KUKA KRL program: EPS_2_251806_MH04A_A_20260212042233.src

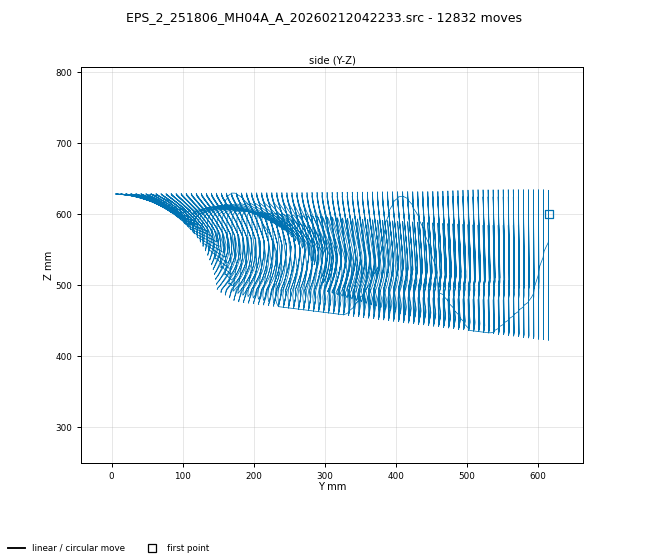
[picture p0: tool path of EPS_2_251806_MH04A_A_20260212042233.src, 12832 of 12834 moves have a stored position in this frame; points joined in program order, loops and branches not executed]
&ACCESS RVP
&REL 4
&COMMENT QRS 19112012
&PARAM EDITMASK = *
DEF PART()
EXT BAS (BAS_COMMAND :IN,REAL :IN )
INT I
BAS (#INITMOV,0 )

;KUKA QRS Post kuka4.cps  Date:22-06-2017 !

File_ID=3012

QRS_PRE_INIT()

;Init var - Until changes are made in qrs_pre_init
Outlet_Square_prg=0
Inlet_1_Square_prg=0
Inlet_2_Square_prg=0
Inlet_3_Square_prg=0
Inlet_4_Square_prg=0
Inlet_5_Square_prg=0

Outlet_1={X 0.000, Y 509.470, Z 509.000, B 0.000, E1 0.000 }
Inlet_1={X 0.000, Y 519.000, Z 484.000, B 0.000, E1 90.000 }
Inlet_2={X 0.000, Y 510.210, Z 499.000, B 0.000, E1 180.000 }
Outlet_1_type=251
Inlet_1_type=201
Inlet_2_type=251
;QRS#1=Sidecore dimensions
;QRS#2=250-10" PVC SDR 35
;QRS#3=200-8" PVC SDR 35
;QRS#4=250-10" PVC SDR 35
;QRS#5=
;QRS#6=
;QRS#7=
;QRS#8=
;QRS#9=14M PSX
;QRS#10=12-08 PSX
;QRS#11=14M PSX
;QRS#12=
;QRS#13=
;QRS#14=
;QRS#15=
;QRS#16=1220x127x914 3'
;QRS#17=EPS Height
;QRS#18=634,5
;QRS#19=*
;QRS#20= UPDATED VERSION 22-06-2017
;QRS#21=*
Outlet_Square=0100
Inlet_1_Square=0100
Inlet_2_Square=0100
Inlet_3_Square=0
Inlet_4_Square=0
Inlet_5_Square=0
Mill_Square=1
Outlet_Square_Prg=205
Inlet_1_Square_prg=204
Inlet_2_Square_prg=205

QRS_INIT()

$ADVANCE=5

; T1
PTP {E1 173.497,E2 173.497}
PTP {X 0,Y 615.499,A -85,B 0,C 180,E1 173.497,E2 173.497,E3 0,E4 0,E5 0,E6 0}
QRS_SPEED_INIT()
LIN {X 0,Y 615.499,Z 600,A -85,B 0,C 180,E1 173.497,E2 173.497,E3 0,E4 0,E5 0,E6 0} C_VEL
LIN {X 0,Y 615.499,Z 575.226,A -85,B 0,C 180,E1 173.497,E2 173.497} C_VEL
LIN {X 0,Y 615.499,Z 564.345,A -85,B 0,C 180,E1 173.497,E2 173.497} C_VEL
LIN {X 0,Y 615.497,Z 562.701,A -85,B 0,C 180,E1 173.417,E2 173.417} C_VEL
LIN {X 0,Y 615.497,Z 555.036,A -85,B 0,C 180,E1 172.455,E2 172.455} C_VEL
LIN {X 0,Y 615.498,Z 545.258,A -85,B 0,C 180,E1 171.463,E2 171.463} C_VEL
LIN {X 0,Y 615.498,Z 534.992,A -85,B 0,C 180,E1 170.636,E2 170.636} C_VEL
LIN {X 0,Y 615.481,Z 523.43,A -85,B 0,C 180,E1 169.889,E2 169.889} C_VEL
LIN {X 0,Y 615.482,Z 511.646,A -85,B 0,C 180,E1 169.296,E2 169.296} C_VEL
LIN {X 0,Y 615.483,Z 498.658,A -85,B 0,C 180,E1 168.807,E2 168.807} C_VEL
LIN {X 0,Y 615.487,Z 486.055,A -85,B 0,C 180,E1 168.473,E2 168.473} C_VEL
LIN {X 0,Y 615.484,Z 478.768,A -85,B 0,C 180,E1 168.327,E2 168.327} C_VEL
LIN {X 0,Y 615.493,Z 471.461,A -85,B 0,C 180,E1 165.451,E2 165.451} C_VEL
LIN {X 0,Y 615.491,Z 464.645,A -85,B 0,C 180,E1 162.729,E2 162.729} C_VEL
LIN {X 0,Y 615.479,Z 457.814,A -85,B 0,C 180,E1 159.967,E2 159.967} C_VEL
LIN {X 0,Y 615.493,Z 452.183,A -85,B 0,C 180,E1 157.654,E2 157.654} C_VEL
LIN {X 0,Y 615.476,Z 445.867,A -85,B 0,C 180,E1 155.008,E2 155.008} C_VEL
LIN {X 0,Y 615.481,Z 440.735,A -85,B 0,C 180,E1 152.822,E2 152.822} C_VEL
LIN {X 0,Y 615.484,Z 434.726,A -85,B 0,C 180,E1 150.207,E2 150.207} C_VEL
LIN {X 0,Y 615.486,Z 428.763,A -85,B 0,C 180,E1 147.542,E2 147.542} C_VEL
LIN {X 0,Y 615.49,Z 422.483,A -85,B 0,C 180,E1 144.685,E2 144.685} C_VEL
LIN {X 0,Y 615.485,Z 422.323,A -85,B 0,C 180,E1 141.931,E2 141.931} C_VEL
LIN {X 0,Y 615.492,Z 422.327,A -85,B 0,C 180,E1 139.394,E2 139.394} C_VEL
LIN {X 0,Y 615.497,Z 422.32,A -85,B 0,C 180,E1 136.756,E2 136.756} C_VEL
LIN {X 0,Y 615.485,Z 422.327,A -85,B 0,C 180,E1 133.997,E2 133.997} C_VEL
LIN {X 0,Y 615.481,Z 422.323,A -85,B 0,C 180,E1 131.093,E2 131.093} C_VEL
LIN {X 0,Y 615.486,Z 422.322,A -85,B 0,C 180,E1 128.905,E2 128.905} C_VEL
LIN {X 0,Y 615.496,Z 422.527,A -85,B 0,C 180,E1 127.626,E2 127.626} C_VEL
LIN {X 0,Y 615.498,Z 431.499,A -85,B 0,C 180,E1 124.702,E2 124.702} C_VEL
LIN {X 0,Y 615.477,Z 438.274,A -85,B 0,C 180,E1 122.329,E2 122.329} C_VEL
LIN {X 0,Y 615.498,Z 445.339,A -85,B 0,C 180,E1 119.796,E2 119.796} C_VEL
LIN {X 0,Y 615.486,Z 453.213,A -85,B 0,C 180,E1 117.044,E2 117.044} C_VEL
LIN {X 0,Y 615.478,Z 461.349,A -85,B 0,C 180,E1 114.273,E2 114.273} C_VEL
LIN {X 0,Y 615.48,Z 469.853,A -85,B 0,C 180,E1 111.433,E2 111.433} C_VEL
LIN {X 0,Y 615.481,Z 478.503,A -85,B 0,C 180,E1 108.602,E2 108.602} C_VEL
LIN {X 0,Y 615.488,Z 486.863,A -85,B 0,C 180,E1 105.906,E2 105.906} C_VEL
LIN {X 0,Y 615.494,Z 492.908,A -85,B 0,C 180,E1 103.993,E2 103.993} C_VEL
LIN {X 0,Y 615.492,Z 507.3,A -85,B 0,C 180,E1 103.748,E2 103.748} C_VEL
LIN {X 0,Y 615.479,Z 521.427,A -85,B 0,C 180,E1 103.37,E2 103.37} C_VEL
LIN {X 0,Y 615.495,Z 535.017,A -85,B 0,C 180,E1 102.866,E2 102.866} C_VEL
LIN {X 0,Y 615.479,Z 547.289,A -85,B 0,C 180,E1 102.28,E2 102.28} C_VEL
LIN {X 0,Y 615.498,Z 559.895,A -85,B 0,C 180,E1 101.527,E2 101.527} C_VEL
LIN {X 0,Y 615.498,Z 571.068,A -85,B 0,C 180,E1 100.709,E2 100.709} C_VEL
LIN {X 0,Y 615.499,Z 580.69,A -85,B 0,C 180,E1 99.863,E2 99.863} C_VEL
LIN {X 0,Y 615.497,Z 590.14,A -85,B 0,C 180,E1 98.868,E2 98.868} C_VEL
LIN {X 0,Y 615.497,Z 599.132,A -85,B 0,C 180,E1 97.711,E2 97.711} C_VEL
LIN {X 0,Y 615.496,Z 606.378,A -85,B 0,C 180,E1 96.557,E2 96.557} C_VEL
LIN {X 0,Y 615.491,Z 612.885,A -85,B 0,C 180,E1 95.242,E2 95.242} C_VEL
LIN {X 0,Y 615.496,Z 617.754,A -85,B 0,C 180,E1 93.929,E2 93.929} C_VEL
LIN {X 0,Y 615.496,Z 621.152,A -85,B 0,C 180,E1 92.619,E2 92.619} C_VEL
LIN {X 0,Y 615.493,Z 623.173,A -85,B 0,C 180,E1 91.309,E2 91.309} C_VEL
LIN {X 0,Y 615.494,Z 623.884,A -85,B 0,C 180,E1 90.001,E2 90.001} C_VEL
LIN {X 0,Y 615.49,Z 623.281,A -85,B 0,C 180,E1 88.692,E2 88.692} C_VEL
LIN {X 0,Y 615.493,Z 621.352,A -85,B 0,C 180,E1 87.383,E2 87.383} C_VEL
LIN {X 0,Y 615.496,Z 618.048,A -85,B 0,C 180,E1 86.072,E2 86.072} C_VEL
LIN {X 0,Y 615.496,Z 613.277,A -85,B 0,C 180,E1 84.76,E2 84.76} C_VEL
LIN {X 0,Y 615.494,Z 606.879,A -85,B 0,C 180,E1 83.444,E2 83.444} C_VEL
LIN {X 0,Y 615.496,Z 599.75,A -85,B 0,C 180,E1 82.29,E2 82.29} C_VEL
LIN {X 0,Y 615.497,Z 592.278,A -85,B 0,C 180,E1 81.299,E2 81.299} C_VEL
LIN {X 0,Y 615.495,Z 583.3,A -85,B 0,C 180,E1 80.305,E2 80.305} C_VEL
LIN {X 0,Y 615.499,Z 572.211,A -85,B 0,C 180,E1 79.291,E2 79.291} C_VEL
LIN {X 0,Y 615.498,Z 561.294,A -85,B 0,C 180,E1 78.474,E2 78.474} C_VEL
LIN {X 0,Y 615.483,Z 549.001,A -85,B 0,C 180,E1 77.722,E2 77.722} C_VEL
LIN {X 0,Y 615.495,Z 537.167,A -85,B 0,C 180,E1 77.136,E2 77.136} C_VEL
LIN {X 0,Y 615.475,Z 524.249,A -85,B 0,C 180,E1 76.631,E2 76.631} C_VEL
LIN {X 0,Y 615.484,Z 511.28,A -85,B 0,C 180,E1 76.253,E2 76.253} C_VEL
LIN {X 0,Y 615.494,Z 497.969,A -85,B 0,C 180,E1 75.987,E2 75.987} C_VEL
LIN {X 0,Y 615.489,Z 492.846,A -85,B 0,C 180,E1 75.911,E2 75.911} C_VEL
LIN {X 0,Y 615.491,Z 483.961,A -85,B 0,C 180,E1 73.073,E2 73.073} C_VEL
LIN {X 0,Y 615.488,Z 475.45,A -85,B 0,C 180,E1 70.316,E2 70.316} C_VEL
LIN {X 0,Y 615.477,Z 467.387,A -85,B 0,C 180,E1 67.657,E2 67.657} C_VEL
LIN {X 0,Y 615.488,Z 459.484,A -85,B 0,C 180,E1 65.009,E2 65.009} C_VEL
LIN {X 0,Y 615.488,Z 450.967,A -85,B 0,C 180,E1 62.086,E2 62.086} C_VEL
LIN {X 0,Y 615.477,Z 443.502,A -85,B 0,C 180,E1 59.462,E2 59.462} C_VEL
LIN {X 0,Y 615.492,Z 436.035,A -85,B 0,C 180,E1 56.765,E2 56.765} C_VEL
LIN {X 0,Y 615.493,Z 428.318,A -85,B 0,C 180,E1 54.166,E2 54.166} C_VEL
LIN {X 0,Y 615.498,Z 422.315,A -85,B 0,C 180,E1 52.183,E2 52.183} C_VEL
LIN {X 0,Y 615.484,Z 422.319,A -85,B 0,C 180,E1 49.395,E2 49.395} C_VEL
LIN {X 0,Y 615.476,Z 422.316,A -85,B 0,C 180,E1 46.756,E2 46.756} C_VEL
LIN {X 0,Y 615.488,Z 422.324,A -85,B 0,C 180,E1 43.999,E2 43.999} C_VEL
LIN {X 0,Y 615.485,Z 422.313,A -85,B 0,C 180,E1 41.474,E2 41.474} C_VEL
LIN {X 0,Y 615.481,Z 422.322,A -85,B 0,C 180,E1 38.905,E2 38.905} C_VEL
LIN {X 0,Y 615.493,Z 422.313,A -85,B 0,C 180,E1 36.425,E2 36.425} C_VEL
LIN {X 0,Y 615.496,Z 422.324,A -85,B 0,C 180,E1 33.538,E2 33.538} C_VEL
LIN {X 0,Y 615.478,Z 422.314,A -85,B 0,C 180,E1 30.92,E2 30.92} C_VEL
LIN {X 0,Y 615.491,Z 422.322,A -85,B 0,C 180,E1 28.454,E2 28.454} C_VEL
LIN {X 0,Y 615.484,Z 422.313,A -85,B 0,C 180,E1 25.571,E2 25.571} C_VEL
LIN {X 0,Y 615.489,Z 422.32,A -85,B 0,C 180,E1 22.845,E2 22.845} C_VEL
LIN {X 0,Y 615.487,Z 422.317,A -85,B 0,C 180,E1 20.033,E2 20.033} C_VEL
LIN {X 0,Y 615.489,Z 422.313,A -85,B 0,C 180,E1 17.271,E2 17.271} C_VEL
LIN {X 0,Y 615.49,Z 422.323,A -85,B 0,C 180,E1 14.549,E2 14.549} C_VEL
LIN {X 0,Y 615.478,Z 422.314,A -85,B 0,C 180,E1 11.861,E2 11.861} C_VEL
LIN {X 0,Y 615.497,Z 422.325,A -85,B 0,C 180,E1 9.199,E2 9.199} C_VEL
LIN {X 0,Y 615.492,Z 422.311,A -85,B 0,C 180,E1 6.557,E2 6.557} C_VEL
LIN {X 0,Y 615.488,Z 422.324,A -85,B 0,C 180,E1 3.929,E2 3.929} C_VEL
LIN {X 0,Y 615.486,Z 422.313,A -85,B 0,C 180,E1 1.309,E2 1.309} C_VEL
LIN {X 0,Y 615.494,Z 422.322,A -85,B 0,C 180,E1 -1.309,E2 -1.309} C_VEL
LIN {X 0,Y 615.476,Z 422.315,A -85,B 0,C 180,E1 -3.929,E2 -3.929} C_VEL
LIN {X 0,Y 615.49,Z 422.32,A -85,B 0,C 180,E1 -6.592,E2 -6.592} C_VEL
LIN {X 0,Y 615.479,Z 422.315,A -85,B 0,C 180,E1 -9.199,E2 -9.199} C_VEL
LIN {X 0,Y 615.478,Z 422.321,A -85,B 0,C 180,E1 -11.861,E2 -11.861} C_VEL
LIN {X 0,Y 615.49,Z 422.315,A -85,B 0,C 180,E1 -14.549,E2 -14.549} C_VEL
LIN {X 0,Y 615.494,Z 422.313,A -85,B 0,C 180,E1 -17.27,E2 -17.27} C_VEL
LIN {X 0,Y 615.489,Z 422.321,A -85,B 0,C 180,E1 -20.033,E2 -20.033} C_VEL
LIN {X 0,Y 615.476,Z 422.315,A -85,B 0,C 180,E1 -22.845,E2 -22.845} C_VEL
LIN {X 0,Y 615.486,Z 422.323,A -85,B 0,C 180,E1 -25.571,E2 -25.571} C_VEL
LIN {X 0,Y 615.492,Z 422.315,A -85,B 0,C 180,E1 -28.454,E2 -28.454} C_VEL
LIN {X 0,Y 615.49,Z 422.315,A -85,B 0,C 180,E1 -31.089,E2 -31.089} C_VEL
LIN {X 0,Y 615.489,Z 422.314,A -85,B 0,C 180,E1 -33.537,E2 -33.537} C_VEL
LIN {X 0,Y 615.488,Z 422.313,A -85,B 0,C 180,E1 -36.425,E2 -36.425} C_VEL
LIN {X 0,Y 615.481,Z 422.322,A -85,B 0,C 180,E1 -39.063,E2 -39.063} C_VEL
LIN {X 0,Y 615.485,Z 422.316,A -85,B 0,C 180,E1 -41.474,E2 -41.474} C_VEL
LIN {X 0,Y 615.491,Z 422.317,A -85,B 0,C 180,E1 -44.149,E2 -44.149} C_VEL
LIN {X 0,Y 615.481,Z 422.314,A -85,B 0,C 180,E1 -46.953,E2 -46.953} C_VEL
LIN {X 0,Y 615.492,Z 422.318,A -85,B 0,C 180,E1 -49.395,E2 -49.395} C_VEL
LIN {X 0,Y 615.484,Z 422.315,A -85,B 0,C 180,E1 -51.989,E2 -51.989} C_VEL
LIN {X 0,Y 615.487,Z 422.315,A -85,B 0,C 180,E1 -54.386,E2 -54.386} C_VEL
LIN {X 0,Y 615.494,Z 422.321,A -85,B 0,C 180,E1 -56.766,E2 -56.766} C_VEL
LIN {X 0,Y 615.484,Z 422.445,A -85,B 0,C 180,E1 -57.954,E2 -57.954} C_VEL
LIN {X 0,Y 615.477,Z 433.27,A -85,B 0,C 180,E1 -60.594,E2 -60.594} C_VEL
LIN {X 0,Y 615.495,Z 444.461,A -85,B 0,C 180,E1 -63.257,E2 -63.257} C_VEL
LIN {X 0,Y 615.482,Z 456.236,A -85,B 0,C 180,E1 -65.993,E2 -65.993} C_VEL
LIN {X 0,Y 615.477,Z 467.542,A -85,B 0,C 180,E1 -68.569,E2 -68.569} C_VEL
LIN {X 0,Y 615.481,Z 480.178,A -85,B 0,C 180,E1 -71.397,E2 -71.397} C_VEL
LIN {X 0,Y 615.485,Z 492.418,A -85,B 0,C 180,E1 -74.096,E2 -74.096} C_VEL
LIN {X 0,Y 615.489,Z 500.83,A -85,B 0,C 180,E1 -75.93,E2 -75.93} C_VEL
LIN {X 0,Y 615.492,Z 515.627,A -85,B 0,C 180,E1 -76.169,E2 -76.169} C_VEL
LIN {X 0,Y 615.486,Z 528.953,A -85,B 0,C 180,E1 -76.506,E2 -76.506} C_VEL
LIN {X 0,Y 615.492,Z 542.169,A -85,B 0,C 180,E1 -76.968,E2 -76.968} C_VEL
LIN {X 0,Y 615.478,Z 555.035,A -85,B 0,C 180,E1 -77.554,E2 -77.554} C_VEL
LIN {X 0,Y 615.497,Z 566.787,A -85,B 0,C 180,E1 -78.224,E2 -78.224} C_VEL
LIN {X 0,Y 615.496,Z 577.419,A -85,B 0,C 180,E1 -78.958,E2 -78.958} C_VEL
LIN {X 0,Y 615.498,Z 587.651,A -85,B 0,C 180,E1 -79.807,E2 -79.807} C_VEL
LIN {X 0,Y 615.498,Z 597.595,A -85,B 0,C 180,E1 -80.802,E2 -80.802} C_VEL
LIN {X 0,Y 615.496,Z 607.079,A -85,B 0,C 180,E1 -81.96,E2 -81.96} C_VEL
LIN {X 0,Y 615.495,Z 614.656,A -85,B 0,C 180,E1 -83.101,E2 -83.101} C_VEL
LIN {X 0,Y 615.494,Z 620.075,A -85,B 0,C 180,E1 -84.102,E2 -84.102} C_VEL
LIN {X 0,Y 615.495,Z 625.686,A -85,B 0,C 180,E1 -85.416,E2 -85.416} C_VEL
LIN {X 0,Y 615.495,Z 629.756,A -85,B 0,C 180,E1 -86.728,E2 -86.728} C_VEL
LIN {X 0,Y 615.497,Z 632.407,A -85,B 0,C 180,E1 -88.038,E2 -88.038} C_VEL
LIN {X 0,Y 615.493,Z 633.723,A -85,B 0,C 180,E1 -89.347,E2 -89.347} C_VEL
LIN {X 0,Y 615.493,Z 633.722,A -85,B 0,C 180,E1 -90.655,E2 -90.655} C_VEL
LIN {X 0,Y 615.498,Z 632.404,A -85,B 0,C 180,E1 -91.964,E2 -91.964} C_VEL
LIN {X 0,Y 615.495,Z 629.752,A -85,B 0,C 180,E1 -93.274,E2 -93.274} C_VEL
LIN {X 0,Y 615.495,Z 625.68,A -85,B 0,C 180,E1 -94.585,E2 -94.585} C_VEL
LIN {X 0,Y 615.494,Z 620.066,A -85,B 0,C 180,E1 -95.899,E2 -95.899} C_VEL
LIN {X 0,Y 615.495,Z 614.651,A -85,B 0,C 180,E1 -96.9,E2 -96.9} C_VEL
LIN {X 0,Y 615.496,Z 607.067,A -85,B 0,C 180,E1 -98.041,E2 -98.041} C_VEL
LIN {X 0,Y 615.498,Z 597.58,A -85,B 0,C 180,E1 -99.199,E2 -99.199} C_VEL
LIN {X 0,Y 615.498,Z 587.633,A -85,B 0,C 180,E1 -100.195,E2 -100.195} C_VEL
LIN {X 0,Y 615.498,Z 576.377,A -85,B 0,C 180,E1 -101.118,E2 -101.118} C_VEL
LIN {X 0,Y 615.496,Z 565.403,A -85,B 0,C 180,E1 -101.861,E2 -101.861} C_VEL
LIN {X 0,Y 615.479,Z 553.314,A -85,B 0,C 180,E1 -102.531,E2 -102.531} C_VEL
LIN {X 0,Y 615.488,Z 539.91,A -85,B 0,C 180,E1 -103.118,E2 -103.118} C_VEL
LIN {X 0,Y 615.488,Z 525.869,A -85,B 0,C 180,E1 -103.58,E2 -103.58} C_VEL
LIN {X 0,Y 615.496,Z 511.604,A -85,B 0,C 180,E1 -103.905,E2 -103.905} C_VEL
LIN {X 0,Y 615.489,Z 500.829,A -85,B 0,C 180,E1 -104.07,E2 -104.07} C_VEL
LIN {X 0,Y 615.494,Z 487.748,A -85,B 0,C 180,E1 -106.929,E2 -106.929} C_VEL
LIN {X 0,Y 615.487,Z 475.313,A -85,B 0,C 180,E1 -109.686,E2 -109.686} C_VEL
LIN {X 0,Y 615.487,Z 462.409,A -85,B 0,C 180,E1 -112.594,E2 -112.594} C_VEL
LIN {X 0,Y 615.477,Z 450.731,A -85,B 0,C 180,E1 -115.28,E2 -115.28} C_VEL
LIN {X 0,Y 615.493,Z 439.498,A -85,B 0,C 180,E1 -117.915,E2 -117.915} C_VEL
LIN {X 0,Y 615.479,Z 428.584,A -85,B 0,C 180,E1 -120.54,E2 -120.54} C_VEL
LIN {X 0,Y 615.482,Z 422.32,A -85,B 0,C 180,E1 -122.087,E2 -122.087} C_VEL
LIN {X 0,Y 615.499,Z 422.319,A -85,B 0,C 180,E1 -124.815,E2 -124.815} C_VEL
LIN {X 0,Y 615.488,Z 422.321,A -85,B 0,C 180,E1 -127.243,E2 -127.243} C_VEL
LIN {X 0,Y 615.483,Z 422.321,A -85,B 0,C 180,E1 -130.088,E2 -130.088} C_VEL
LIN {X 0,Y 615.491,Z 422.319,A -85,B 0,C 180,E1 -133.048,E2 -133.048} C_VEL
LIN {X 0,Y 615.488,Z 422.32,A -85,B 0,C 180,E1 -136.003,E2 -136.003} C_VEL
LIN {X 0,Y 615.492,Z 422.319,A -85,B 0,C 180,E1 -138.906,E2 -138.906} C_VEL
LIN {X 0,Y 615.49,Z 422.321,A -85,B 0,C 180,E1 -141.932,E2 -141.932} C_VEL
LIN {X 0,Y 615.495,Z 422.386,A -85,B 0,C 180,E1 -144.886,E2 -144.886} C_VEL
LIN {X 0,Y 615.493,Z 428.829,A -85,B 0,C 180,E1 -147.669,E2 -147.669} C_VEL
LIN {X 0,Y 615.492,Z 435.398,A -85,B 0,C 180,E1 -150.594,E2 -150.594} C_VEL
LIN {X 0,Y 615.48,Z 440.839,A -85,B 0,C 180,E1 -152.957,E2 -152.957} C_VEL
LIN {X 0,Y 615.493,Z 447.354,A -85,B 0,C 180,E1 -155.728,E2 -155.728} C_VEL
LIN {X 0,Y 615.494,Z 454.183,A -85,B 0,C 180,E1 -158.568,E2 -158.568} C_VEL
LIN {X 0,Y 615.484,Z 461.112,A -85,B 0,C 180,E1 -161.397,E2 -161.397} C_VEL
LIN {X 0,Y 615.476,Z 467.832,A -85,B 0,C 180,E1 -164.095,E2 -164.095} C_VEL
LIN {X 0,Y 615.497,Z 474.644,A -85,B 0,C 180,E1 -166.799,E2 -166.799} C_VEL
LIN {X 0,Y 615.485,Z 478.804,A -85,B 0,C 180,E1 -168.431,E2 -168.431} C_VEL
LIN {X 0,Y 615.495,Z 491.197,A -85,B 0,C 180,E1 -168.682,E2 -168.682} C_VEL
LIN {X 0,Y 615.48,Z 503.99,A -85,B 0,C 180,E1 -169.079,E2 -169.079} C_VEL
LIN {X 0,Y 615.498,Z 515.321,A -85,B 0,C 180,E1 -169.556,E2 -169.556} C_VEL
LIN {X 0,Y 615.479,Z 526.127,A -85,B 0,C 180,E1 -170.138,E2 -170.138} C_VEL
LIN {X 0,Y 615.498,Z 537.159,A -85,B 0,C 180,E1 -170.884,E2 -170.884} C_VEL
LIN {X 0,Y 615.498,Z 547.831,A -85,B 0,C 180,E1 -171.794,E2 -171.794} C_VEL
LIN {X 0,Y 615.498,Z 555.709,A -85,B 0,C 180,E1 -172.62,E2 -172.62} C_VEL
LIN {X 0,Y 615.497,Z 563.399,A -85,B 0,C 180,E1 -173.608,E2 -173.608} C_VEL
LIN {X 0,Y 615.498,Z 570.458,A -85,B 0,C 180,E1 -174.759,E2 -174.759} C_VEL
LIN {X 0,Y 615.493,Z 575.158,A -85,B 0,C 180,E1 -175.744,E2 -175.744} C_VEL
LIN {X 0,Y 615.496,Z 578.754,A -85,B 0,C 180,E1 -176.727,E2 -176.727} C_VEL
LIN {X 0,Y 615.496,Z 580.615,A -85,B 0,C 180,E1 -177.382,E2 -177.382} C_VEL
LIN {X 0,Y 615.497,Z 582.034,A -85,B 0,C 180,E1 -178.037,E2 -178.037} C_VEL
LIN {X 0,Y 615.496,Z 583.642,A -85,B 0,C 180,E1 -179.346,E2 -179.346} C_VEL
LIN {X 0,Y 615.494,Z 583.884,A -85,B 0,C 180,E1 -180,E2 -180} C_VEL
LIN {X 0,Y 615.496,Z 583.705,A -85,B 0,C 180,E1 -180.654,E2 -180.654} C_VEL
LIN {X 0,Y 615.496,Z 582.183,A -85,B 0,C 180,E1 -181.963,E2 -181.963} C_VEL
LIN {X 0,Y 615.498,Z 580.841,A -85,B 0,C 180,E1 -182.618,E2 -182.618} C_VEL
LIN {X 0,Y 615.497,Z 577.994,A -85,B 0,C 180,E1 -183.601,E2 -183.601} C_VEL
LIN {X 0,Y 615.499,Z 574.134,A -85,B 0,C 180,E1 -184.585,E2 -184.585} C_VEL
LIN {X 0,Y 615.498,Z 569.151,A -85,B 0,C 180,E1 -185.57,E2 -185.57} C_VEL
LIN {X 0,Y 615.497,Z 562.701,A -85,B 0,C 180,E1 -186.583,E2 -186.583} C_VEL
LIN {X 0,Y 614.829,Z 559.519,A -85,B 0,C 180,E1 -187.032,E2 -187.032} C_VEL
LIN {X 0,Y 611.988,Z 553.946,A -85,B 0,C 180,E1 -187.749,E2 -187.749} C_VEL
LIN {X 0,Y 609.138,Z 547.669,A -85,B 0,C 180,E1 -188.43,E2 -188.43} C_VEL
LIN {X 0,Y 608.477,Z 543.428,A -85,B 0,C 180,E1 -188.82,E2 -188.82} C_VEL
LIN {X 0,Y 608.494,Z 532.889,A -85,B 0,C 180,E1 -189.641,E2 -189.641} C_VEL
LIN {X 0,Y 608.49,Z 522.11,A -85,B 0,C 180,E1 -190.313,E2 -190.313} C_VEL
LIN {X 0,Y 608.511,Z 509.505,A -85,B 0,C 180,E1 -190.925,E2 -190.925} C_VEL
LIN {X 0,Y 608.522,Z 497.464,A -85,B 0,C 180,E1 -191.365,E2 -191.365} C_VEL
LIN {X 0,Y 608.545,Z 485.153,A -85,B 0,C 180,E1 -191.681,E2 -191.681} C_VEL
LIN {X 0,Y 608.441,Z 479.165,A -85,B 0,C 180,E1 -191.81,E2 -191.81} C_VEL
LIN {X 0,Y 608.45,Z 471.814,A -85,B 0,C 180,E1 -194.721,E2 -194.721} C_VEL
LIN {X 0,Y 608.434,Z 464.946,A -85,B 0,C 180,E1 -197.477,E2 -197.477} C_VEL
LIN {X 0,Y 608.443,Z 458.078,A -85,B 0,C 180,E1 -200.275,E2 -200.275} C_VEL
LIN {X 0,Y 608.447,Z 451.209,A -85,B 0,C 180,E1 -203.124,E2 -203.124} C_VEL
LIN {X 0,Y 608.448,Z 445.088,A -85,B 0,C 180,E1 -205.715,E2 -205.715} C_VEL
LIN {X 0,Y 608.448,Z 439.189,A -85,B 0,C 180,E1 -208.267,E2 -208.267} C_VEL
LIN {X 0,Y 608.451,Z 434.037,A -85,B 0,C 180,E1 -210.546,E2 -210.546} C_VEL
LIN {X 0,Y 608.462,Z 428.867,A -85,B 0,C 180,E1 -212.879,E2 -212.879} C_VEL
LIN {X 0,Y 608.454,Z 423.321,A -85,B 0,C 180,E1 -215.48,E2 -215.48} C_VEL
LIN {X 0,Y 608.467,Z 423.32,A -85,B 0,C 180,E1 -218.24,E2 -218.24} C_VEL
LIN {X 0,Y 608.463,Z 423.319,A -85,B 0,C 180,E1 -221.342,E2 -221.342} C_VEL
LIN {X 0,Y 608.465,Z 423.319,A -85,B 0,C 180,E1 -224.264,E2 -224.264} C_VEL
LIN {X 0,Y 608.447,Z 423.323,A -85,B 0,C 180,E1 -227.039,E2 -227.039} C_VEL
LIN {X 0,Y 608.458,Z 423.32,A -85,B 0,C 180,E1 -229.696,E2 -229.696} C_VEL
LIN {X 0,Y 608.491,Z 423.52,A -85,B 0,C 180,E1 -232.336,E2 -232.336} C_VEL
LIN {X 0,Y 608.491,Z 431.902,A -85,B 0,C 180,E1 -235.089,E2 -235.089} C_VEL
LIN {X 0,Y 608.483,Z 438.94,A -85,B 0,C 180,E1 -237.475,E2 -237.475} C_VEL
LIN {X 0,Y 608.483,Z 446.528,A -85,B 0,C 180,E1 -240.221,E2 -240.221} C_VEL
LIN {X 0,Y 608.481,Z 453.829,A -85,B 0,C 180,E1 -242.793,E2 -242.793} C_VEL
LIN {X 0,Y 608.461,Z 461.49,A -85,B 0,C 180,E1 -245.429,E2 -245.429} C_VEL
LIN {X 0,Y 608.459,Z 470.04,A -85,B 0,C 180,E1 -248.307,E2 -248.307} C_VEL
LIN {X 0,Y 608.464,Z 478.59,A -85,B 0,C 180,E1 -251.13,E2 -251.13} C_VEL
LIN {X 0,Y 608.442,Z 487.141,A -85,B 0,C 180,E1 -253.905,E2 -253.905} C_VEL
LIN {X 0,Y 608.445,Z 493.296,A -85,B 0,C 180,E1 -255.846,E2 -255.846} C_VEL
LIN {X 0,Y 608.598,Z 507.877,A -85,B 0,C 180,E1 -256.106,E2 -256.106} C_VEL
LIN {X 0,Y 608.565,Z 521.461,A -85,B 0,C 180,E1 -256.475,E2 -256.475} C_VEL
LIN {X 0,Y 608.558,Z 535.068,A -85,B 0,C 180,E1 -256.985,E2 -256.985} C_VEL
LIN {X 0,Y 608.528,Z 547.36,A -85,B 0,C 180,E1 -257.578,E2 -257.578} C_VEL
LIN {X 0,Y 608.524,Z 560.003,A -85,B 0,C 180,E1 -258.339,E2 -258.339} C_VEL
LIN {X 0,Y 608.505,Z 571.616,A -85,B 0,C 180,E1 -259.197,E2 -259.197} C_VEL
LIN {X 0,Y 608.488,Z 582.635,A -85,B 0,C 180,E1 -260.19,E2 -260.19} C_VEL
LIN {X 0,Y 608.476,Z 591.825,A -85,B 0,C 180,E1 -261.196,E2 -261.196} C_VEL
LIN {X 0,Y 608.452,Z 600.612,A -85,B 0,C 180,E1 -262.366,E2 -262.366} C_VEL
LIN {X 0,Y 608.452,Z 608.237,A -85,B 0,C 180,E1 -263.63,E2 -263.63} C_VEL
LIN {X 0,Y 608.436,Z 613.371,A -85,B 0,C 180,E1 -264.697,E2 -264.697} C_VEL
LIN {X 0,Y 608.434,Z 618.294,A -85,B 0,C 180,E1 -266.025,E2 -266.025} C_VEL
LIN {X 0,Y 608.425,Z 621.732,A -85,B 0,C 180,E1 -267.351,E2 -267.351} C_VEL
LIN {X 0,Y 608.446,Z 623.777,A -85,B 0,C 180,E1 -268.675,E2 -268.675} C_VEL
LIN {X 0,Y 608.434,Z 624.495,A -85,B 0,C 180,E1 -269.999,E2 -269.999} C_VEL
LIN {X 0,Y 608.443,Z 623.883,A -85,B 0,C 180,E1 -271.323,E2 -271.323} C_VEL
LIN {X 0,Y 608.421,Z 621.93,A -85,B 0,C 180,E1 -272.647,E2 -272.647} C_VEL
LIN {X 0,Y 608.434,Z 618.587,A -85,B 0,C 180,E1 -273.973,E2 -273.973} C_VEL
LIN {X 0,Y 608.44,Z 613.763,A -85,B 0,C 180,E1 -275.301,E2 -275.301} C_VEL
LIN {X 0,Y 608.442,Z 607.478,A -85,B 0,C 180,E1 -276.6,E2 -276.6} C_VEL
LIN {X 0,Y 608.453,Z 600.106,A -85,B 0,C 180,E1 -277.799,E2 -277.799} C_VEL
LIN {X 0,Y 608.476,Z 592.57,A -85,B 0,C 180,E1 -278.802,E2 -278.802} C_VEL
LIN {X 0,Y 608.486,Z 583.524,A -85,B 0,C 180,E1 -279.808,E2 -279.808} C_VEL
LIN {X 0,Y 608.507,Z 572.724,A -85,B 0,C 180,E1 -280.804,E2 -280.804} C_VEL
LIN {X 0,Y 608.523,Z 561.39,A -85,B 0,C 180,E1 -281.66,E2 -281.66} C_VEL
LIN {X 0,Y 608.53,Z 549.056,A -85,B 0,C 180,E1 -282.421,E2 -282.421} C_VEL
LIN {X 0,Y 608.556,Z 537.196,A -85,B 0,C 180,E1 -283.014,E2 -283.014} C_VEL
LIN {X 0,Y 608.559,Z 524.251,A -85,B 0,C 180,E1 -283.523,E2 -283.523} C_VEL
LIN {X 0,Y 608.592,Z 510.013,A -85,B 0,C 180,E1 -283.935,E2 -283.935} C_VEL
LIN {X 0,Y 608.605,Z 495.722,A -85,B 0,C 180,E1 -284.206,E2 -284.206} C_VEL
LIN {X 0,Y 608.45,Z 493.121,A -85,B 0,C 180,E1 -284.267,E2 -284.267} C_VEL
LIN {X 0,Y 608.443,Z 484.218,A -85,B 0,C 180,E1 -287.129,E2 -287.129} C_VEL
LIN {X 0,Y 608.452,Z 475.663,A -85,B 0,C 180,E1 -289.921,E2 -289.921} C_VEL
LIN {X 0,Y 608.457,Z 467.966,A -85,B 0,C 180,E1 -292.475,E2 -292.475} C_VEL
LIN {X 0,Y 608.459,Z 459.621,A -85,B 0,C 180,E1 -295.299,E2 -295.299} C_VEL
LIN {X 0,Y 608.468,Z 452.134,A -85,B 0,C 180,E1 -297.89,E2 -297.89} C_VEL
LIN {X 0,Y 608.474,Z 444.647,A -85,B 0,C 180,E1 -300.543,E2 -300.543} C_VEL
LIN {X 0,Y 608.49,Z 437.129,A -85,B 0,C 180,E1 -303.271,E2 -303.271} C_VEL
LIN {X 0,Y 608.476,Z 428.594,A -85,B 0,C 180,E1 -306.089,E2 -306.089} C_VEL
LIN {X 0,Y 608.485,Z 423.314,A -85,B 0,C 180,E1 -307.867,E2 -307.867} C_VEL
LIN {X 0,Y 608.445,Z 423.317,A -85,B 0,C 180,E1 -310.328,E2 -310.328} C_VEL
LIN {X 0,Y 608.448,Z 423.319,A -85,B 0,C 180,E1 -312.959,E2 -312.959} C_VEL
LIN {X 0,Y 608.462,Z 423.316,A -85,B 0,C 180,E1 -315.734,E2 -315.734} C_VEL
LIN {X 0,Y 608.459,Z 423.314,A -85,B 0,C 180,E1 -318.656,E2 -318.656} C_VEL
LIN {X 0,Y 608.465,Z 423.32,A -85,B 0,C 180,E1 -321.411,E2 -321.411} C_VEL
LIN {X 0,Y 608.47,Z 423.313,A -85,B 0,C 180,E1 -323.949,E2 -323.949} C_VEL
LIN {X 0,Y 608.47,Z 423.318,A -85,B 0,C 180,E1 -326.33,E2 -326.33} C_VEL
LIN {X 0,Y 608.471,Z 423.314,A -85,B 0,C 180,E1 -328.726,E2 -328.726} C_VEL
LIN {X 0,Y 608.471,Z 423.316,A -85,B 0,C 180,E1 -331.378,E2 -331.378} C_VEL
LIN {X 0,Y 608.444,Z 423.317,A -85,B 0,C 180,E1 -333.964,E2 -333.964} C_VEL
LIN {X 0,Y 608.46,Z 423.314,A -85,B 0,C 180,E1 -336.155,E2 -336.155} C_VEL
LIN {X 0,Y 608.469,Z 423.316,A -85,B 0,C 180,E1 -338.308,E2 -338.308} C_VEL
LIN {X 0,Y 608.465,Z 423.313,A -85,B 0,C 180,E1 -341.282,E2 -341.282} C_VEL
LIN {X 0,Y 608.46,Z 423.321,A -85,B 0,C 180,E1 -343.906,E2 -343.906} C_VEL
LIN {X 0,Y 608.459,Z 423.314,A -85,B 0,C 180,E1 -346.643,E2 -346.643} C_VEL
LIN {X 0,Y 608.471,Z 423.316,A -85,B 0,C 180,E1 -349.35,E2 -349.35} C_VEL
LIN {X 0,Y 608.47,Z 423.314,A -85,B 0,C 180,E1 -352.033,E2 -352.033} C_VEL
LIN {X 0,Y 608.464,Z 423.315,A -85,B 0,C 180,E1 -354.698,E2 -354.698} C_VEL
LIN {X 0,Y 608.479,Z 423.315,A -85,B 0,C 180,E1 -357.352,E2 -357.352} C_VEL
LIN {X 0,Y 608.468,Z 423.314,A -85,B 0,C 180,E1 -360,E2 -360} C_VEL
LIN {X 0,Y 608.482,Z 423.315,A -85,B 0,C 180,E1 -362.648,E2 -362.648} C_VEL
LIN {X 0,Y 608.465,Z 423.314,A -85,B 0,C 180,E1 -365.302,E2 -365.302} C_VEL
LIN {X 0,Y 608.48,Z 423.318,A -85,B 0,C 180,E1 -367.967,E2 -367.967} C_VEL
LIN {X 0,Y 608.461,Z 423.314,A -85,B 0,C 180,E1 -370.959,E2 -370.959} C_VEL
LIN {X 0,Y 608.463,Z 423.321,A -85,B 0,C 180,E1 -373.356,E2 -373.356} C_VEL
LIN {X 0,Y 608.456,Z 423.315,A -85,B 0,C 180,E1 -376.094,E2 -376.094} C_VEL
LIN {X 0,Y 608.453,Z 423.317,A -85,B 0,C 180,E1 -378.87,E2 -378.87} C_VEL
LIN {X 0,Y 608.473,Z 423.316,A -85,B 0,C 180,E1 -381.691,E2 -381.691} C_VEL
LIN {X 0,Y 608.45,Z 423.315,A -85,B 0,C 180,E1 -384.571,E2 -384.571} C_VEL
LIN {X 0,Y 608.478,Z 423.319,A -85,B 0,C 180,E1 -387.21,E2 -387.21} C_VEL
LIN {X 0,Y 608.461,Z 423.314,A -85,B 0,C 180,E1 -389.973,E2 -389.973} C_VEL
LIN {X 0,Y 608.464,Z 423.319,A -85,B 0,C 180,E1 -392.525,E2 -392.525} C_VEL
LIN {X 0,Y 608.443,Z 423.317,A -85,B 0,C 180,E1 -395.278,E2 -395.278} C_VEL
LIN {X 0,Y 608.467,Z 423.318,A -85,B 0,C 180,E1 -397.746,E2 -397.746} C_VEL
LIN {X 0,Y 608.474,Z 423.313,A -85,B 0,C 180,E1 -400.333,E2 -400.333} C_VEL
LIN {X 0,Y 608.483,Z 423.312,A -85,B 0,C 180,E1 -403.312,E2 -403.312} C_VEL
LIN {X 0,Y 608.467,Z 423.32,A -85,B 0,C 180,E1 -406.132,E2 -406.132} C_VEL
LIN {X 0,Y 608.45,Z 423.315,A -85,B 0,C 180,E1 -408.825,E2 -408.825} C_VEL
LIN {X 0,Y 608.468,Z 423.321,A -85,B 0,C 180,E1 -411.413,E2 -411.413} C_VEL
LIN {X 0,Y 608.474,Z 423.312,A -85,B 0,C 180,E1 -413.951,E2 -413.951} C_VEL
LIN {X 0,Y 608.462,Z 423.318,A -85,B 0,C 180,E1 -416.331,E2 -416.331} C_VEL
LIN {X 0,Y 608.476,Z 423.487,A -85,B 0,C 180,E1 -417.801,E2 -417.801} C_VEL
LIN {X 0,Y 608.539,Z 433.279,A -85,B 0,C 180,E1 -420.226,E2 -420.226} C_VEL
LIN {X 0,Y 608.517,Z 443.9,A -85,B 0,C 180,E1 -422.786,E2 -422.786} C_VEL
LIN {X 0,Y 608.52,Z 455.134,A -85,B 0,C 180,E1 -425.433,E2 -425.433} C_VEL
LIN {X 0,Y 608.479,Z 467.623,A -85,B 0,C 180,E1 -428.31,E2 -428.31} C_VEL
LIN {X 0,Y 608.462,Z 480.112,A -85,B 0,C 180,E1 -431.132,E2 -431.132} C_VEL
LIN {X 0,Y 608.463,Z 492.6,A -85,B 0,C 180,E1 -433.907,E2 -433.907} C_VEL
LIN {X 0,Y 608.443,Z 501.089,A -85,B 0,C 180,E1 -435.771,E2 -435.771} C_VEL
LIN {X 0,Y 608.591,Z 516.26,A -85,B 0,C 180,E1 -436.023,E2 -436.023} C_VEL
LIN {X 0,Y 608.584,Z 530.289,A -85,B 0,C 180,E1 -436.392,E2 -436.392} C_VEL
LIN {X 0,Y 608.552,Z 542.196,A -85,B 0,C 180,E1 -436.817,E2 -436.817} C_VEL
LIN {X 0,Y 608.517,Z 555.09,A -85,B 0,C 180,E1 -437.41,E2 -437.41} C_VEL
LIN {X 0,Y 608.534,Z 568.161,A -85,B 0,C 180,E1 -438.172,E2 -438.172} C_VEL
LIN {X 0,Y 608.506,Z 580.046,A -85,B 0,C 180,E1 -439.027,E2 -439.027} C_VEL
LIN {X 0,Y 608.472,Z 591.4,A -85,B 0,C 180,E1 -440.024,E2 -440.024} C_VEL
LIN {X 0,Y 608.472,Z 600.831,A -85,B 0,C 180,E1 -441.03,E2 -441.03} C_VEL
LIN {X 0,Y 608.453,Z 609.803,A -85,B 0,C 180,E1 -442.201,E2 -442.201} C_VEL
LIN {X 0,Y 608.441,Z 617.231,A -85,B 0,C 180,E1 -443.4,E2 -443.4} C_VEL
LIN {X 0,Y 608.44,Z 623.571,A -85,B 0,C 180,E1 -444.699,E2 -444.699} C_VEL
LIN {X 0,Y 608.431,Z 628.444,A -85,B 0,C 180,E1 -446.027,E2 -446.027} C_VEL
LIN {X 0,Y 608.424,Z 631.833,A -85,B 0,C 180,E1 -447.353,E2 -447.353} C_VEL
LIN {X 0,Y 608.442,Z 633.831,A -85,B 0,C 180,E1 -448.677,E2 -448.677} C_VEL
LIN {X 0,Y 608.433,Z 634.5,A -85,B 0,C 180,E1 -450.001,E2 -450.001} C_VEL
LIN {X 0,Y 608.442,Z 633.829,A -85,B 0,C 180,E1 -451.325,E2 -451.325} C_VEL
LIN {X 0,Y 608.424,Z 631.829,A -85,B 0,C 180,E1 -452.649,E2 -452.649} C_VEL
LIN {X 0,Y 608.431,Z 628.439,A -85,B 0,C 180,E1 -453.975,E2 -453.975} C_VEL
LIN {X 0,Y 608.44,Z 623.564,A -85,B 0,C 180,E1 -455.303,E2 -455.303} C_VEL
LIN {X 0,Y 608.446,Z 617.207,A -85,B 0,C 180,E1 -456.604,E2 -456.604} C_VEL
LIN {X 0,Y 608.453,Z 609.792,A -85,B 0,C 180,E1 -457.801,E2 -457.801} C_VEL
LIN {X 0,Y 608.473,Z 600.816,A -85,B 0,C 180,E1 -458.971,E2 -458.971} C_VEL
LIN {X 0,Y 608.472,Z 591.382,A -85,B 0,C 180,E1 -459.978,E2 -459.978} C_VEL
LIN {X 0,Y 608.506,Z 580.044,A -85,B 0,C 180,E1 -460.973,E2 -460.973} C_VEL
LIN {X 0,Y 608.534,Z 568.136,A -85,B 0,C 180,E1 -461.83,E2 -461.83} C_VEL
LIN {X 0,Y 608.517,Z 555.058,A -85,B 0,C 180,E1 -462.592,E2 -462.592} C_VEL
LIN {X 0,Y 608.553,Z 542.153,A -85,B 0,C 180,E1 -463.185,E2 -463.185} C_VEL
LIN {X 0,Y 608.588,Z 528.153,A -85,B 0,C 180,E1 -463.673,E2 -463.673} C_VEL
LIN {X 0,Y 608.6,Z 514.411,A -85,B 0,C 180,E1 -464.014,E2 -464.014} C_VEL
LIN {X 0,Y 608.442,Z 501.096,A -85,B 0,C 180,E1 -464.227,E2 -464.227} C_VEL
LIN {X 0,Y 608.485,Z 487.909,A -85,B 0,C 180,E1 -467.13,E2 -467.13} C_VEL
LIN {X 0,Y 608.487,Z 475.42,A -85,B 0,C 180,E1 -469.922,E2 -469.922} C_VEL
LIN {X 0,Y 608.51,Z 462.933,A -85,B 0,C 180,E1 -472.763,E2 -472.763} C_VEL
LIN {X 0,Y 608.504,Z 452.004,A -85,B 0,C 180,E1 -475.299,E2 -475.299} C_VEL
LIN {X 0,Y 608.53,Z 441.077,A -85,B 0,C 180,E1 -477.888,E2 -477.888} C_VEL
LIN {X 0,Y 608.542,Z 430.149,A -85,B 0,C 180,E1 -480.541,E2 -480.541} C_VEL
LIN {X 0,Y 608.461,Z 423.318,A -85,B 0,C 180,E1 -482.255,E2 -482.255} C_VEL
LIN {X 0,Y 608.488,Z 423.315,A -85,B 0,C 180,E1 -484.911,E2 -484.911} C_VEL
LIN {X 0,Y 608.47,Z 423.318,A -85,B 0,C 180,E1 -487.747,E2 -487.747} C_VEL
LIN {X 0,Y 608.453,Z 423.322,A -85,B 0,C 180,E1 -490.329,E2 -490.329} C_VEL
LIN {X 0,Y 608.481,Z 423.319,A -85,B 0,C 180,E1 -493.31,E2 -493.31} C_VEL
LIN {X 0,Y 608.474,Z 423.318,A -85,B 0,C 180,E1 -496.131,E2 -496.131} C_VEL
LIN {X 0,Y 608.46,Z 423.318,A -85,B 0,C 180,E1 -498.824,E2 -498.824} C_VEL
LIN {X 0,Y 608.47,Z 423.316,A -85,B 0,C 180,E1 -501.76,E2 -501.76} C_VEL
LIN {X 0,Y 608.461,Z 423.318,A -85,B 0,C 180,E1 -504.723,E2 -504.723} C_VEL
LIN {X 0,Y 608.49,Z 423.894,A -85,B 0,C 180,E1 -505.09,E2 -505.09} C_VEL
LIN {X 0,Y 608.473,Z 430.383,A -85,B 0,C 180,E1 -507.906,E2 -507.906} C_VEL
LIN {X 0,Y 608.484,Z 435.552,A -85,B 0,C 180,E1 -510.221,E2 -510.221} C_VEL
LIN {X 0,Y 608.457,Z 441.425,A -85,B 0,C 180,E1 -512.797,E2 -512.797} C_VEL
LIN {X 0,Y 608.453,Z 447.563,A -85,B 0,C 180,E1 -515.429,E2 -515.429} C_VEL
LIN {X 0,Y 608.447,Z 454.427,A -85,B 0,C 180,E1 -518.308,E2 -518.308} C_VEL
LIN {X 0,Y 608.435,Z 461.292,A -85,B 0,C 180,E1 -521.13,E2 -521.13} C_VEL
LIN {X 0,Y 608.441,Z 468.156,A -85,B 0,C 180,E1 -523.906,E2 -523.906} C_VEL
LIN {X 0,Y 608.435,Z 475.021,A -85,B 0,C 180,E1 -526.643,E2 -526.643} C_VEL
LIN {X 0,Y 608.435,Z 479.205,A -85,B 0,C 180,E1 -528.296,E2 -528.296} C_VEL
LIN {X 0,Y 608.551,Z 492.855,A -85,B 0,C 180,E1 -528.593,E2 -528.593} C_VEL
LIN {X 0,Y 608.501,Z 506.223,A -85,B 0,C 180,E1 -529.031,E2 -529.031} C_VEL
LIN {X 0,Y 608.513,Z 517.235,A -85,B 0,C 180,E1 -529.519,E2 -529.519} C_VEL
LIN {X 0,Y 608.472,Z 529.013,A -85,B 0,C 180,E1 -530.191,E2 -530.191} C_VEL
LIN {X 0,Y 608.485,Z 539.525,A -85,B 0,C 180,E1 -530.946,E2 -530.946} C_VEL
LIN {X 0,Y 608.475,Z 548.134,A -85,B 0,C 180,E1 -531.699,E2 -531.699} C_VEL
LIN {X 0,Y 608.471,Z 556.064,A -85,B 0,C 180,E1 -532.534,E2 -532.534} C_VEL
LIN {X 0,Y 608.468,Z 563.571,A -85,B 0,C 180,E1 -533.498,E2 -533.498} C_VEL
LIN {X 0,Y 608.451,Z 569.11,A -85,B 0,C 180,E1 -534.366,E2 -534.366} C_VEL
LIN {X 0,Y 608.431,Z 574.252,A -85,B 0,C 180,E1 -535.362,E2 -535.362} C_VEL
LIN {X 0,Y 608.45,Z 578.241,A -85,B 0,C 180,E1 -536.358,E2 -536.358} C_VEL
LIN {X 0,Y 608.425,Z 581.191,A -85,B 0,C 180,E1 -537.352,E2 -537.352} C_VEL
LIN {X 0,Y 608.442,Z 582.627,A -85,B 0,C 180,E1 -538.014,E2 -538.014} C_VEL
LIN {X 0,Y 608.439,Z 584.252,A -85,B 0,C 180,E1 -539.338,E2 -539.338} C_VEL
LIN {X 0,Y 608.434,Z 584.495,A -85,B 0,C 180,E1 -540,E2 -540} C_VEL
LIN {X 0,Y 608.439,Z 584.315,A -85,B 0,C 180,E1 -540.662,E2 -540.662} C_VEL
LIN {X 0,Y 608.441,Z 582.776,A -85,B 0,C 180,E1 -541.986,E2 -541.986} C_VEL
LIN {X 0,Y 608.426,Z 581.418,A -85,B 0,C 180,E1 -542.648,E2 -542.648} C_VEL
LIN {X 0,Y 608.45,Z 578.541,A -85,B 0,C 180,E1 -543.642,E2 -543.642} C_VEL
LIN {X 0,Y 608.433,Z 574.642,A -85,B 0,C 180,E1 -544.638,E2 -544.638} C_VEL
LIN {X 0,Y 608.449,Z 569.612,A -85,B 0,C 180,E1 -545.634,E2 -545.634} C_VEL
LIN {X 0,Y 608.442,Z 563.294,A -85,B 0,C 180,E1 -546.633,E2 -546.633} C_VEL
LIN {X 0,Y 608.475,Z 555.378,A -85,B 0,C 180,E1 -547.633,E2 -547.633} C_VEL
LIN {X 0,Y 608.472,Z 545.535,A -85,B 0,C 180,E1 -548.636,E2 -548.636} C_VEL
LIN {X 0,Y 608.477,Z 543.428,A -85,B 0,C 180,E1 -548.82,E2 -548.82} C_VEL
LIN {X 0,Y 607.803,Z 539.094,A -85,B 0,C 180,E1 -549.19,E2 -549.19} C_VEL
LIN {X 0,Y 604.94,Z 531.847,A -85,B 0,C 180,E1 -549.77,E2 -549.77} C_VEL
LIN {X 0,Y 602.126,Z 524.205,A -85,B 0,C 180,E1 -550.302,E2 -550.302} C_VEL
LIN {X 0,Y 601.531,Z 519.138,A -85,B 0,C 180,E1 -550.595,E2 -550.595} C_VEL
LIN {X 0,Y 601.539,Z 507.392,A -85,B 0,C 180,E1 -551.144,E2 -551.144} C_VEL
LIN {X 0,Y 601.578,Z 494.555,A -85,B 0,C 180,E1 -551.584,E2 -551.584} C_VEL
LIN {X 0,Y 601.591,Z 481.703,A -85,B 0,C 180,E1 -551.882,E2 -551.882} C_VEL
LIN {X 0,Y 601.342,Z 479.163,A -85,B 0,C 180,E1 -551.952,E2 -551.952} C_VEL
LIN {X 0,Y 601.367,Z 471.813,A -85,B 0,C 180,E1 -554.899,E2 -554.899} C_VEL
LIN {X 0,Y 601.362,Z 464.945,A -85,B 0,C 180,E1 -557.689,E2 -557.689} C_VEL
LIN {X 0,Y 601.37,Z 458.077,A -85,B 0,C 180,E1 -560.524,E2 -560.524} C_VEL
LIN {X 0,Y 601.379,Z 451.208,A -85,B 0,C 180,E1 -563.412,E2 -563.412} C_VEL
LIN {X 0,Y 601.383,Z 445.501,A -85,B 0,C 180,E1 -565.86,E2 -565.86} C_VEL
LIN {X 0,Y 601.413,Z 438.836,A -85,B 0,C 180,E1 -568.784,E2 -568.784} C_VEL
LIN {X 0,Y 601.407,Z 432.304,A -85,B 0,C 180,E1 -571.727,E2 -571.727} C_VEL
LIN {X 0,Y 601.434,Z 427.106,A -85,B 0,C 180,E1 -574.118,E2 -574.118} C_VEL
LIN {X 0,Y 601.423,Z 424.197,A -85,B 0,C 180,E1 -575.579,E2 -575.579} C_VEL
LIN {X 0,Y 601.418,Z 424.199,A -85,B 0,C 180,E1 -578.469,E2 -578.469} C_VEL
LIN {X 0,Y 601.418,Z 424.197,A -85,B 0,C 180,E1 -580.874,E2 -580.874} C_VEL
LIN {X 0,Y 601.455,Z 424.192,A -85,B 0,C 180,E1 -583.584,E2 -583.584} C_VEL
LIN {X 0,Y 601.433,Z 424.195,A -85,B 0,C 180,E1 -586.427,E2 -586.427} C_VEL
LIN {X 0,Y 601.415,Z 424.199,A -85,B 0,C 180,E1 -589.427,E2 -589.427} C_VEL
LIN {X 0,Y 601.442,Z 424.31,A -85,B 0,C 180,E1 -592.264,E2 -592.264} C_VEL
LIN {X 0,Y 601.448,Z 432.756,A -85,B 0,C 180,E1 -595.07,E2 -595.07} C_VEL
LIN {X 0,Y 601.474,Z 441.164,A -85,B 0,C 180,E1 -597.882,E2 -597.882} C_VEL
LIN {X 0,Y 601.479,Z 448.667,A -85,B 0,C 180,E1 -600.609,E2 -600.609} C_VEL
LIN {X 0,Y 601.424,Z 456.148,A -85,B 0,C 180,E1 -603.262,E2 -603.262} C_VEL
LIN {X 0,Y 601.432,Z 463.629,A -85,B 0,C 180,E1 -605.858,E2 -605.858} C_VEL
LIN {X 0,Y 601.408,Z 472.179,A -85,B 0,C 180,E1 -608.76,E2 -608.76} C_VEL
LIN {X 0,Y 601.399,Z 480.73,A -85,B 0,C 180,E1 -611.607,E2 -611.607} C_VEL
LIN {X 0,Y 601.366,Z 489.281,A -85,B 0,C 180,E1 -614.407,E2 -614.407} C_VEL
LIN {X 0,Y 601.363,Z 493.142,A -85,B 0,C 180,E1 -615.659,E2 -615.659} C_VEL
LIN {X 0,Y 601.738,Z 496.597,A -85,B 0,C 180,E1 -615.732,E2 -615.732} C_VEL
LIN {X 0,Y 601.683,Z 510.702,A -85,B 0,C 180,E1 -616.009,E2 -616.009} C_VEL
LIN {X 0,Y 601.647,Z 524.605,A -85,B 0,C 180,E1 -616.42,E2 -616.42} C_VEL
LIN {X 0,Y 601.624,Z 537.056,A -85,B 0,C 180,E1 -616.918,E2 -616.918} C_VEL
LIN {X 0,Y 601.563,Z 548.937,A -85,B 0,C 180,E1 -617.517,E2 -617.517} C_VEL
LIN {X 0,Y 601.535,Z 561.281,A -85,B 0,C 180,E1 -618.287,E2 -618.287} C_VEL
LIN {X 0,Y 601.496,Z 572.303,A -85,B 0,C 180,E1 -619.124,E2 -619.124} C_VEL
LIN {X 0,Y 601.435,Z 582.635,A -85,B 0,C 180,E1 -620.074,E2 -620.074} C_VEL
LIN {X 0,Y 601.411,Z 591.829,A -85,B 0,C 180,E1 -621.092,E2 -621.092} C_VEL
LIN {X 0,Y 601.387,Z 600.618,A -85,B 0,C 180,E1 -622.276,E2 -622.276} C_VEL
LIN {X 0,Y 601.374,Z 607.382,A -85,B 0,C 180,E1 -623.395,E2 -623.395} C_VEL
LIN {X 0,Y 601.352,Z 613.373,A -85,B 0,C 180,E1 -624.634,E2 -624.634} C_VEL
LIN {X 0,Y 601.345,Z 618.294,A -85,B 0,C 180,E1 -625.978,E2 -625.978} C_VEL
LIN {X 0,Y 601.324,Z 621.735,A -85,B 0,C 180,E1 -627.32,E2 -627.32} C_VEL
LIN {X 0,Y 601.346,Z 623.78,A -85,B 0,C 180,E1 -628.66,E2 -628.66} C_VEL
LIN {X 0,Y 601.334,Z 624.492,A -85,B 0,C 180,E1 -629.999,E2 -629.999} C_VEL
LIN {X 0,Y 601.342,Z 623.882,A -85,B 0,C 180,E1 -631.339,E2 -631.339} C_VEL
LIN {X 0,Y 601.321,Z 621.931,A -85,B 0,C 180,E1 -632.679,E2 -632.679} C_VEL
LIN {X 0,Y 601.346,Z 618.583,A -85,B 0,C 180,E1 -634.02,E2 -634.02} C_VEL
LIN {X 0,Y 601.355,Z 613.761,A -85,B 0,C 180,E1 -635.364,E2 -635.364} C_VEL
LIN {X 0,Y 601.355,Z 607.301,A -85,B 0,C 180,E1 -636.711,E2 -636.711} C_VEL
LIN {X 0,Y 601.399,Z 600.105,A -85,B 0,C 180,E1 -637.891,E2 -637.891} C_VEL
LIN {X 0,Y 601.411,Z 592.565,A -85,B 0,C 180,E1 -638.906,E2 -638.906} C_VEL
LIN {X 0,Y 601.431,Z 583.513,A -85,B 0,C 180,E1 -639.924,E2 -639.924} C_VEL
LIN {X 0,Y 601.497,Z 573.35,A -85,B 0,C 180,E1 -640.876,E2 -640.876} C_VEL
LIN {X 0,Y 601.549,Z 561.375,A -85,B 0,C 180,E1 -641.797,E2 -641.797} C_VEL
LIN {X 0,Y 601.577,Z 549.047,A -85,B 0,C 180,E1 -642.566,E2 -642.566} C_VEL
LIN {X 0,Y 601.622,Z 537.19,A -85,B 0,C 180,E1 -643.166,E2 -643.166} C_VEL
LIN {X 0,Y 601.664,Z 523.251,A -85,B 0,C 180,E1 -643.714,E2 -643.714} C_VEL
LIN {X 0,Y 601.694,Z 509.388,A -85,B 0,C 180,E1 -644.112,E2 -644.112} C_VEL
LIN {X 0,Y 601.633,Z 494.835,A -85,B 0,C 180,E1 -644.386,E2 -644.386} C_VEL
LIN {X 0,Y 601.366,Z 493.119,A -85,B 0,C 180,E1 -644.439,E2 -644.439} C_VEL
LIN {X 0,Y 601.386,Z 484.216,A -85,B 0,C 180,E1 -647.337,E2 -647.337} C_VEL
LIN {X 0,Y 601.39,Z 475.661,A -85,B 0,C 180,E1 -650.165,E2 -650.165} C_VEL
LIN {X 0,Y 601.424,Z 467.105,A -85,B 0,C 180,E1 -653.045,E2 -653.045} C_VEL
LIN {X 0,Y 601.428,Z 458.89,A -85,B 0,C 180,E1 -655.87,E2 -655.87} C_VEL
LIN {X 0,Y 601.445,Z 451.062,A -85,B 0,C 180,E1 -658.625,E2 -658.625} C_VEL
LIN {X 0,Y 601.486,Z 443.202,A -85,B 0,C 180,E1 -661.465,E2 -661.465} C_VEL
LIN {X 0,Y 601.433,Z 435.477,A -85,B 0,C 180,E1 -664.117,E2 -664.117} C_VEL
LIN {X 0,Y 601.439,Z 426.891,A -85,B 0,C 180,E1 -666.981,E2 -666.981} C_VEL
LIN {X 0,Y 601.443,Z 424.191,A -85,B 0,C 180,E1 -667.893,E2 -667.893} C_VEL
LIN {X 0,Y 601.412,Z 424.195,A -85,B 0,C 180,E1 -670.573,E2 -670.573} C_VEL
LIN {X 0,Y 601.443,Z 424.188,A -85,B 0,C 180,E1 -673.583,E2 -673.583} C_VEL
LIN {X 0,Y 601.444,Z 424.192,A -85,B 0,C 180,E1 -676.424,E2 -676.424} C_VEL
LIN {X 0,Y 601.413,Z 424.198,A -85,B 0,C 180,E1 -679.425,E2 -679.425} C_VEL
LIN {X 0,Y 601.419,Z 424.193,A -85,B 0,C 180,E1 -681.732,E2 -681.732} C_VEL
LIN {X 0,Y 601.4,Z 424.195,A -85,B 0,C 180,E1 -684.246,E2 -684.246} C_VEL
LIN {X 0,Y 601.429,Z 424.195,A -85,B 0,C 180,E1 -686.686,E2 -686.686} C_VEL
LIN {X 0,Y 601.426,Z 424.19,A -85,B 0,C 180,E1 -689.058,E2 -689.058} C_VEL
LIN {X 0,Y 601.43,Z 424.193,A -85,B 0,C 180,E1 -691.373,E2 -691.373} C_VEL
LIN {X 0,Y 601.402,Z 424.198,A -85,B 0,C 180,E1 -693.636,E2 -693.636} C_VEL
LIN {X 0,Y 601.417,Z 424.195,A -85,B 0,C 180,E1 -696.589,E2 -696.589} C_VEL
LIN {X 0,Y 601.429,Z 424.19,A -85,B 0,C 180,E1 -699.478,E2 -699.478} C_VEL
LIN {X 0,Y 601.403,Z 424.198,A -85,B 0,C 180,E1 -702.312,E2 -702.312} C_VEL
LIN {X 0,Y 601.413,Z 424.193,A -85,B 0,C 180,E1 -704.409,E2 -704.409} C_VEL
LIN {X 0,Y 601.423,Z 424.197,A -85,B 0,C 180,E1 -707.172,E2 -707.172} C_VEL
LIN {X 0,Y 601.43,Z 424.19,A -85,B 0,C 180,E1 -709.905,E2 -709.905} C_VEL
LIN {X 0,Y 601.445,Z 424.194,A -85,B 0,C 180,E1 -712.615,E2 -712.615} C_VEL
LIN {X 0,Y 601.423,Z 424.191,A -85,B 0,C 180,E1 -715.308,E2 -715.308} C_VEL
LIN {X 0,Y 601.418,Z 424.195,A -85,B 0,C 180,E1 -717.991,E2 -717.991} C_VEL
LIN {X 0,Y 601.447,Z 424.189,A -85,B 0,C 180,E1 -720.669,E2 -720.669} C_VEL
LIN {X 0,Y 601.432,Z 424.19,A -85,B 0,C 180,E1 -723.349,E2 -723.349} C_VEL
LIN {X 0,Y 601.409,Z 424.195,A -85,B 0,C 180,E1 -726.037,E2 -726.037} C_VEL
LIN {X 0,Y 601.433,Z 424.19,A -85,B 0,C 180,E1 -728.738,E2 -728.738} C_VEL
LIN {X 0,Y 601.427,Z 424.196,A -85,B 0,C 180,E1 -731.458,E2 -731.458} C_VEL
LIN {X 0,Y 601.41,Z 424.192,A -85,B 0,C 180,E1 -734.206,E2 -734.206} C_VEL
LIN {X 0,Y 601.428,Z 424.194,A -85,B 0,C 180,E1 -736.986,E2 -736.986} C_VEL
LIN {X 0,Y 601.406,Z 424.195,A -85,B 0,C 180,E1 -739.809,E2 -739.809} C_VEL
LIN {X 0,Y 601.41,Z 424.192,A -85,B 0,C 180,E1 -742.683,E2 -742.683} C_VEL
LIN {X 0,Y 601.398,Z 424.195,A -85,B 0,C 180,E1 -744.879,E2 -744.879} C_VEL
LIN {X 0,Y 601.418,Z 424.191,A -85,B 0,C 180,E1 -747.868,E2 -747.868} C_VEL
LIN {X 0,Y 601.439,Z 424.19,A -85,B 0,C 180,E1 -750.163,E2 -750.163} C_VEL
LIN {X 0,Y 601.424,Z 424.193,A -85,B 0,C 180,E1 -752.718,E2 -752.718} C_VEL
LIN {X 0,Y 601.407,Z 424.193,A -85,B 0,C 180,E1 -755.116,E2 -755.116} C_VEL
LIN {X 0,Y 601.429,Z 424.196,A -85,B 0,C 180,E1 -757.42,E2 -757.42} C_VEL
LIN {X 0,Y 601.406,Z 424.193,A -85,B 0,C 180,E1 -759.996,E2 -759.996} C_VEL
LIN {X 0,Y 601.434,Z 424.196,A -85,B 0,C 180,E1 -762.668,E2 -762.668} C_VEL
LIN {X 0,Y 601.418,Z 424.191,A -85,B 0,C 180,E1 -765.483,E2 -765.483} C_VEL
LIN {X 0,Y 601.422,Z 424.193,A -85,B 0,C 180,E1 -768.407,E2 -768.407} C_VEL
LIN {X 0,Y 601.433,Z 424.191,A -85,B 0,C 180,E1 -770.877,E2 -770.877} C_VEL
LIN {X 0,Y 601.439,Z 424.19,A -85,B 0,C 180,E1 -773.735,E2 -773.735} C_VEL
LIN {X 0,Y 601.431,Z 424.192,A -85,B 0,C 180,E1 -776.065,E2 -776.065} C_VEL
LIN {X 0,Y 601.435,Z 424.308,A -85,B 0,C 180,E1 -777.585,E2 -777.585} C_VEL
LIN {X 0,Y 601.61,Z 429.044,A -85,B 0,C 180,E1 -778.792,E2 -778.792} C_VEL
LIN {X 0,Y 601.572,Z 439.523,A -85,B 0,C 180,E1 -781.382,E2 -781.382} C_VEL
LIN {X 0,Y 601.525,Z 450.848,A -85,B 0,C 180,E1 -784.111,E2 -784.111} C_VEL
LIN {X 0,Y 601.5,Z 462.94,A -85,B 0,C 180,E1 -786.958,E2 -786.958} C_VEL
LIN {X 0,Y 601.464,Z 475.428,A -85,B 0,C 180,E1 -789.837,E2 -789.837} C_VEL
LIN {X 0,Y 601.437,Z 487.917,A -85,B 0,C 180,E1 -792.665,E2 -792.665} C_VEL
LIN {X 0,Y 601.389,Z 500.913,A -85,B 0,C 180,E1 -795.562,E2 -795.562} C_VEL
LIN {X 0,Y 601.381,Z 501.089,A -85,B 0,C 180,E1 -795.6,E2 -795.6} C_VEL
LIN {X 0,Y 601.749,Z 505.389,A -85,B 0,C 180,E1 -795.67,E2 -795.67} C_VEL
LIN {X 0,Y 601.723,Z 519.849,A -85,B 0,C 180,E1 -795.945,E2 -795.945} C_VEL
LIN {X 0,Y 601.67,Z 533.941,A -85,B 0,C 180,E1 -796.354,E2 -796.354} C_VEL
LIN {X 0,Y 601.626,Z 546.15,A -85,B 0,C 180,E1 -796.834,E2 -796.834} C_VEL
LIN {X 0,Y 601.564,Z 559.793,A -85,B 0,C 180,E1 -797.519,E2 -797.519} C_VEL
LIN {X 0,Y 601.534,Z 571.984,A -85,B 0,C 180,E1 -798.289,E2 -798.289} C_VEL
LIN {X 0,Y 601.486,Z 582.763,A -85,B 0,C 180,E1 -799.118,E2 -799.118} C_VEL
LIN {X 0,Y 601.432,Z 593.09,A -85,B 0,C 180,E1 -800.076,E2 -800.076} C_VEL
LIN {X 0,Y 601.411,Z 602.205,A -85,B 0,C 180,E1 -801.094,E2 -801.094} C_VEL
LIN {X 0,Y 601.385,Z 610.925,A -85,B 0,C 180,E1 -802.277,E2 -802.277} C_VEL
LIN {X 0,Y 601.367,Z 617.648,A -85,B 0,C 180,E1 -803.399,E2 -803.399} C_VEL
LIN {X 0,Y 601.355,Z 623.571,A -85,B 0,C 180,E1 -804.636,E2 -804.636} C_VEL
LIN {X 0,Y 601.343,Z 628.444,A -85,B 0,C 180,E1 -805.98,E2 -805.98} C_VEL
LIN {X 0,Y 601.323,Z 631.833,A -85,B 0,C 180,E1 -807.321,E2 -807.321} C_VEL
LIN {X 0,Y 601.342,Z 633.832,A -85,B 0,C 180,E1 -808.661,E2 -808.661} C_VEL
LIN {X 0,Y 601.333,Z 634.5,A -85,B 0,C 180,E1 -810.001,E2 -810.001} C_VEL
LIN {X 0,Y 601.342,Z 633.83,A -85,B 0,C 180,E1 -811.34,E2 -811.34} C_VEL
LIN {X 0,Y 601.324,Z 631.83,A -85,B 0,C 180,E1 -812.68,E2 -812.68} C_VEL
LIN {X 0,Y 601.343,Z 628.439,A -85,B 0,C 180,E1 -814.022,E2 -814.022} C_VEL
LIN {X 0,Y 601.355,Z 623.564,A -85,B 0,C 180,E1 -815.366,E2 -815.366} C_VEL
LIN {X 0,Y 601.356,Z 617.047,A -85,B 0,C 180,E1 -816.712,E2 -816.712} C_VEL
LIN {X 0,Y 601.398,Z 609.793,A -85,B 0,C 180,E1 -817.893,E2 -817.893} C_VEL
LIN {X 0,Y 601.43,Z 600.816,A -85,B 0,C 180,E1 -819.077,E2 -819.077} C_VEL
LIN {X 0,Y 601.44,Z 591.383,A -85,B 0,C 180,E1 -820.096,E2 -820.096} C_VEL
LIN {X 0,Y 601.505,Z 580.689,A -85,B 0,C 180,E1 -821.051,E2 -821.051} C_VEL
LIN {X 0,Y 601.546,Z 569.414,A -85,B 0,C 180,E1 -821.884,E2 -821.884} C_VEL
LIN {X 0,Y 601.551,Z 556.629,A -85,B 0,C 180,E1 -822.654,E2 -822.654} C_VEL
LIN {X 0,Y 601.622,Z 544.14,A -85,B 0,C 180,E1 -823.254,E2 -823.254} C_VEL
LIN {X 0,Y 601.681,Z 530.824,A -85,B 0,C 180,E1 -823.749,E2 -823.749} C_VEL
LIN {X 0,Y 601.717,Z 516.815,A -85,B 0,C 180,E1 -824.127,E2 -824.127} C_VEL
LIN {X 0,Y 601.656,Z 502.63,A -85,B 0,C 180,E1 -824.372,E2 -824.372} C_VEL
LIN {X 0,Y 601.402,Z 501.043,A -85,B 0,C 180,E1 -824.409,E2 -824.409} C_VEL
LIN {X 0,Y 601.438,Z 487.909,A -85,B 0,C 180,E1 -827.337,E2 -827.337} C_VEL
LIN {X 0,Y 601.465,Z 475.42,A -85,B 0,C 180,E1 -830.164,E2 -830.164} C_VEL
LIN {X 0,Y 601.502,Z 462.932,A -85,B 0,C 180,E1 -833.043,E2 -833.043} C_VEL
LIN {X 0,Y 601.528,Z 450.845,A -85,B 0,C 180,E1 -835.89,E2 -835.89} C_VEL
LIN {X 0,Y 601.575,Z 438.728,A -85,B 0,C 180,E1 -838.813,E2 -838.813} C_VEL
LIN {X 0,Y 601.634,Z 427.926,A -85,B 0,C 180,E1 -841.488,E2 -841.488} C_VEL
LIN {X 0,Y 601.415,Z 424.198,A -85,B 0,C 180,E1 -842.468,E2 -842.468} C_VEL
LIN {X 0,Y 601.419,Z 424.195,A -85,B 0,C 180,E1 -845.115,E2 -845.115} C_VEL
LIN {X 0,Y 601.439,Z 424.196,A -85,B 0,C 180,E1 -847.419,E2 -847.419} C_VEL
LIN {X 0,Y 601.416,Z 424.195,A -85,B 0,C 180,E1 -849.995,E2 -849.995} C_VEL
LIN {X 0,Y 601.413,Z 424.194,A -85,B 0,C 180,E1 -852.671,E2 -852.671} C_VEL
LIN {X 0,Y 601.431,Z 424.192,A -85,B 0,C 180,E1 -855.482,E2 -855.482} C_VEL
LIN {X 0,Y 601.428,Z 424.193,A -85,B 0,C 180,E1 -858.407,E2 -858.407} C_VEL
LIN {X 0,Y 601.407,Z 424.199,A -85,B 0,C 180,E1 -860.873,E2 -860.873} C_VEL
LIN {X 0,Y 601.401,Z 424.199,A -85,B 0,C 180,E1 -863.417,E2 -863.417} C_VEL
LIN {X 0,Y 601.453,Z 424.339,A -85,B 0,C 180,E1 -864.881,E2 -864.881} C_VEL
LIN {X 0,Y 601.435,Z 430.31,A -85,B 0,C 180,E1 -867.484,E2 -867.484} C_VEL
LIN {X 0,Y 601.409,Z 435.599,A -85,B 0,C 180,E1 -869.856,E2 -869.856} C_VEL
LIN {X 0,Y 601.382,Z 440.701,A -85,B 0,C 180,E1 -872.131,E2 -872.131} C_VEL
LIN {X 0,Y 601.415,Z 445.849,A -85,B 0,C 180,E1 -874.382,E2 -874.382} C_VEL
LIN {X 0,Y 601.386,Z 452.917,A -85,B 0,C 180,E1 -877.403,E2 -877.403} C_VEL
LIN {X 0,Y 601.378,Z 459.577,A -85,B 0,C 180,E1 -880.19,E2 -880.19} C_VEL
LIN {X 0,Y 601.36,Z 466.441,A -85,B 0,C 180,E1 -883.012,E2 -883.012} C_VEL
LIN {X 0,Y 601.349,Z 473.665,A -85,B 0,C 180,E1 -885.937,E2 -885.937} C_VEL
LIN {X 0,Y 601.342,Z 479.206,A -85,B 0,C 180,E1 -888.156,E2 -888.156} C_VEL
LIN {X 0,Y 601.625,Z 488.669,A -85,B 0,C 180,E1 -888.353,E2 -888.353} C_VEL
LIN {X 0,Y 601.569,Z 501.908,A -85,B 0,C 180,E1 -888.739,E2 -888.739} C_VEL
LIN {X 0,Y 601.519,Z 513.751,A -85,B 0,C 180,E1 -889.226,E2 -889.226} C_VEL
LIN {X 0,Y 601.491,Z 524.922,A -85,B 0,C 180,E1 -889.821,E2 -889.821} C_VEL
LIN {X 0,Y 601.455,Z 536.299,A -85,B 0,C 180,E1 -890.585,E2 -890.585} C_VEL
LIN {X 0,Y 601.424,Z 546.365,A -85,B 0,C 180,E1 -891.432,E2 -891.432} C_VEL
LIN {X 0,Y 601.418,Z 556.069,A -85,B 0,C 180,E1 -892.446,E2 -892.446} C_VEL
LIN {X 0,Y 601.377,Z 563.391,A -85,B 0,C 180,E1 -893.393,E2 -893.393} C_VEL
LIN {X 0,Y 601.372,Z 569.113,A -85,B 0,C 180,E1 -894.299,E2 -894.299} C_VEL
LIN {X 0,Y 601.335,Z 574.254,A -85,B 0,C 180,E1 -895.307,E2 -895.307} C_VEL
LIN {X 0,Y 601.368,Z 578.243,A -85,B 0,C 180,E1 -896.315,E2 -896.315} C_VEL
LIN {X 0,Y 601.324,Z 581.193,A -85,B 0,C 180,E1 -897.32,E2 -897.32} C_VEL
LIN {X 0,Y 601.341,Z 582.627,A -85,B 0,C 180,E1 -897.991,E2 -897.991} C_VEL
LIN {X 0,Y 601.339,Z 584.253,A -85,B 0,C 180,E1 -899.33,E2 -899.33} C_VEL
LIN {X 0,Y 601.335,Z 584.496,A -85,B 0,C 180,E1 -900,E2 -900} C_VEL
LIN {X 0,Y 601.339,Z 584.315,A -85,B 0,C 180,E1 -900.67,E2 -900.67} C_VEL
LIN {X 0,Y 601.34,Z 582.775,A -85,B 0,C 180,E1 -902.009,E2 -902.009} C_VEL
LIN {X 0,Y 601.326,Z 581.417,A -85,B 0,C 180,E1 -902.68,E2 -902.68} C_VEL
LIN {X 0,Y 601.368,Z 578.54,A -85,B 0,C 180,E1 -903.685,E2 -903.685} C_VEL
LIN {X 0,Y 601.337,Z 574.64,A -85,B 0,C 180,E1 -904.693,E2 -904.693} C_VEL
LIN {X 0,Y 601.373,Z 569.609,A -85,B 0,C 180,E1 -905.701,E2 -905.701} C_VEL
LIN {X 0,Y 601.383,Z 563.291,A -85,B 0,C 180,E1 -906.711,E2 -906.711} C_VEL
LIN {X 0,Y 601.396,Z 555.373,A -85,B 0,C 180,E1 -907.723,E2 -907.723} C_VEL
LIN {X 0,Y 601.437,Z 545.529,A -85,B 0,C 180,E1 -908.738,E2 -908.738} C_VEL
LIN {X 0,Y 601.449,Z 535.207,A -85,B 0,C 180,E1 -909.585,E2 -909.585} C_VEL
LIN {X 0,Y 601.493,Z 523.588,A -85,B 0,C 180,E1 -910.349,E2 -910.349} C_VEL
LIN {X 0,Y 601.531,Z 519.138,A -85,B 0,C 180,E1 -910.595,E2 -910.595} C_VEL
LIN {X 0,Y 600.95,Z 514.009,A -85,B 0,C 180,E1 -910.868,E2 -910.868} C_VEL
LIN {X 0,Y 598.191,Z 505.557,A -85,B 0,C 180,E1 -911.287,E2 -911.287} C_VEL
LIN {X 0,Y 595.358,Z 496.813,A -85,B 0,C 180,E1 -911.642,E2 -911.642} C_VEL
LIN {X 0,Y 594.657,Z 491.228,A -85,B 0,C 180,E1 -911.814,E2 -911.814} C_VEL
LIN {X 0,Y 594.449,Z 480.533,A -85,B 0,C 180,E1 -912.049,E2 -912.049} C_VEL
LIN {X 0,Y 594.255,Z 479.162,A -85,B 0,C 180,E1 -912.096,E2 -912.096} C_VEL
LIN {X 0,Y 594.281,Z 471.811,A -85,B 0,C 180,E1 -915.08,E2 -915.08} C_VEL
LIN {X 0,Y 594.292,Z 466.66,A -85,B 0,C 180,E1 -917.196,E2 -917.196} C_VEL
LIN {X 0,Y 594.292,Z 461.509,A -85,B 0,C 180,E1 -919.337,E2 -919.337} C_VEL
LIN {X 0,Y 594.319,Z 454.641,A -85,B 0,C 180,E1 -922.235,E2 -922.235} C_VEL
LIN {X 0,Y 594.328,Z 447.772,A -85,B 0,C 180,E1 -925.195,E2 -925.195} C_VEL
LIN {X 0,Y 594.346,Z 442.495,A -85,B 0,C 180,E1 -927.518,E2 -927.518} C_VEL
LIN {X 0,Y 594.375,Z 436.275,A -85,B 0,C 180,E1 -930.325,E2 -930.325} C_VEL
LIN {X 0,Y 594.386,Z 430.567,A -85,B 0,C 180,E1 -932.95,E2 -932.95} C_VEL
LIN {X 0,Y 594.388,Z 425.073,A -85,B 0,C 180,E1 -935.563,E2 -935.563} C_VEL
LIN {X 0,Y 594.387,Z 425.072,A -85,B 0,C 180,E1 -937.941,E2 -937.941} C_VEL
LIN {X 0,Y 594.381,Z 425.074,A -85,B 0,C 180,E1 -940.822,E2 -940.822} C_VEL
LIN {X 0,Y 594.389,Z 425.075,A -85,B 0,C 180,E1 -943.841,E2 -943.841} C_VEL
LIN {X 0,Y 594.369,Z 425.075,A -85,B 0,C 180,E1 -946.7,E2 -946.7} C_VEL
LIN {X 0,Y 594.37,Z 425.077,A -85,B 0,C 180,E1 -949.432,E2 -949.432} C_VEL
LIN {X 0,Y 594.423,Z 425.173,A -85,B 0,C 180,E1 -952.207,E2 -952.207} C_VEL
LIN {X 0,Y 594.399,Z 432.515,A -85,B 0,C 180,E1 -954.67,E2 -954.67} C_VEL
LIN {X 0,Y 594.402,Z 440.761,A -85,B 0,C 180,E1 -957.467,E2 -957.467} C_VEL
LIN {X 0,Y 594.46,Z 447.12,A -85,B 0,C 180,E1 -959.66,E2 -959.66} C_VEL
LIN {X 0,Y 594.423,Z 455.081,A -85,B 0,C 180,E1 -962.541,E2 -962.541} C_VEL
LIN {X 0,Y 594.381,Z 462.562,A -85,B 0,C 180,E1 -965.18,E2 -965.18} C_VEL
LIN {X 0,Y 594.347,Z 470.044,A -85,B 0,C 180,E1 -967.765,E2 -967.765} C_VEL
LIN {X 0,Y 594.332,Z 478.594,A -85,B 0,C 180,E1 -970.664,E2 -970.664} C_VEL
LIN {X 0,Y 594.304,Z 487.145,A -85,B 0,C 180,E1 -973.511,E2 -973.511} C_VEL
LIN {X 0,Y 594.293,Z 493.163,A -85,B 0,C 180,E1 -975.49,E2 -975.49} C_VEL
LIN {X 0,Y 594.867,Z 497.054,A -85,B 0,C 180,E1 -975.569,E2 -975.569} C_VEL
LIN {X 0,Y 594.802,Z 511.064,A -85,B 0,C 180,E1 -975.852,E2 -975.852} C_VEL
LIN {X 0,Y 594.75,Z 524.789,A -85,B 0,C 180,E1 -976.265,E2 -976.265} C_VEL
LIN {X 0,Y 594.711,Z 537.075,A -85,B 0,C 180,E1 -976.763,E2 -976.763} C_VEL
LIN {X 0,Y 594.607,Z 548.948,A -85,B 0,C 180,E1 -977.369,E2 -977.369} C_VEL
LIN {X 0,Y 594.548,Z 561.283,A -85,B 0,C 180,E1 -978.147,E2 -978.147} C_VEL
LIN {X 0,Y 594.481,Z 572.155,A -85,B 0,C 180,E1 -978.982,E2 -978.982} C_VEL
LIN {X 0,Y 594.414,Z 582.635,A -85,B 0,C 180,E1 -979.956,E2 -979.956} C_VEL
LIN {X 0,Y 594.369,Z 591.831,A -85,B 0,C 180,E1 -980.985,E2 -980.985} C_VEL
LIN {X 0,Y 594.317,Z 600.624,A -85,B 0,C 180,E1 -982.183,E2 -982.183} C_VEL
LIN {X 0,Y 594.301,Z 607.798,A -85,B 0,C 180,E1 -983.393,E2 -983.393} C_VEL
LIN {X 0,Y 594.273,Z 613.375,A -85,B 0,C 180,E1 -984.57,E2 -984.57} C_VEL
LIN {X 0,Y 594.261,Z 618.294,A -85,B 0,C 180,E1 -985.93,E2 -985.93} C_VEL
LIN {X 0,Y 594.224,Z 621.737,A -85,B 0,C 180,E1 -987.288,E2 -987.288} C_VEL
LIN {X 0,Y 594.245,Z 623.783,A -85,B 0,C 180,E1 -988.644,E2 -988.644} C_VEL
LIN {X 0,Y 594.235,Z 624.486,A -85,B 0,C 180,E1 -989.999,E2 -989.999} C_VEL
LIN {X 0,Y 594.242,Z 623.879,A -85,B 0,C 180,E1 -991.355,E2 -991.355} C_VEL
LIN {X 0,Y 594.221,Z 621.931,A -85,B 0,C 180,E1 -992.711,E2 -992.711} C_VEL
LIN {X 0,Y 594.262,Z 618.579,A -85,B 0,C 180,E1 -994.068,E2 -994.068} C_VEL
LIN {X 0,Y 594.275,Z 613.758,A -85,B 0,C 180,E1 -995.428,E2 -995.428} C_VEL
LIN {X 0,Y 594.277,Z 607.301,A -85,B 0,C 180,E1 -996.791,E2 -996.791} C_VEL
LIN {X 0,Y 594.329,Z 600.104,A -85,B 0,C 180,E1 -997.986,E2 -997.986} C_VEL
LIN {X 0,Y 594.368,Z 592.56,A -85,B 0,C 180,E1 -999.013,E2 -999.013} C_VEL
LIN {X 0,Y 594.399,Z 583.503,A -85,B 0,C 180,E1 -1000.043,E2 -1000.043} C_VEL
LIN {X 0,Y 594.477,Z 573.229,A -85,B 0,C 180,E1 -1001.016,E2 -1001.016} C_VEL
LIN {X 0,Y 594.571,Z 561.36,A -85,B 0,C 180,E1 -1001.937,E2 -1001.937} C_VEL
LIN {X 0,Y 594.604,Z 549.038,A -85,B 0,C 180,E1 -1002.716,E2 -1002.716} C_VEL
LIN {X 0,Y 594.682,Z 537.183,A -85,B 0,C 180,E1 -1003.323,E2 -1003.323} C_VEL
LIN {X 0,Y 594.764,Z 523.583,A -85,B 0,C 180,E1 -1003.865,E2 -1003.865} C_VEL
LIN {X 0,Y 594.804,Z 510.055,A -85,B 0,C 180,E1 -1004.262,E2 -1004.262} C_VEL
LIN {X 0,Y 594.854,Z 496.222,A -85,B 0,C 180,E1 -1004.533,E2 -1004.533} C_VEL
LIN {X 0,Y 594.308,Z 493.138,A -85,B 0,C 180,E1 -1004.607,E2 -1004.607} C_VEL
LIN {X 0,Y 594.32,Z 484.214,A -85,B 0,C 180,E1 -1007.549,E2 -1007.549} C_VEL
LIN {X 0,Y 594.356,Z 475.659,A -85,B 0,C 180,E1 -1010.414,E2 -1010.414} C_VEL
LIN {X 0,Y 594.368,Z 467.103,A -85,B 0,C 180,E1 -1013.334,E2 -1013.334} C_VEL
LIN {X 0,Y 594.401,Z 459.38,A -85,B 0,C 180,E1 -1016.025,E2 -1016.025} C_VEL
LIN {X 0,Y 594.451,Z 451.06,A -85,B 0,C 180,E1 -1018.993,E2 -1018.993} C_VEL
LIN {X 0,Y 594.454,Z 443.623,A -85,B 0,C 180,E1 -1021.654,E2 -1021.654} C_VEL
LIN {X 0,Y 594.412,Z 435.027,A -85,B 0,C 180,E1 -1024.576,E2 -1024.576} C_VEL
LIN {X 0,Y 594.43,Z 427.585,A -85,B 0,C 180,E1 -1027.082,E2 -1027.082} C_VEL
LIN {X 0,Y 594.409,Z 425.068,A -85,B 0,C 180,E1 -1027.937,E2 -1027.937} C_VEL
LIN {X 0,Y 594.376,Z 425.076,A -85,B 0,C 180,E1 -1030.822,E2 -1030.822} C_VEL
LIN {X 0,Y 594.376,Z 425.07,A -85,B 0,C 180,E1 -1033.84,E2 -1033.84} C_VEL
LIN {X 0,Y 594.38,Z 425.069,A -85,B 0,C 180,E1 -1036.702,E2 -1036.702} C_VEL
LIN {X 0,Y 594.367,Z 425.075,A -85,B 0,C 180,E1 -1039.433,E2 -1039.433} C_VEL
LIN {X 0,Y 594.385,Z 425.068,A -85,B 0,C 180,E1 -1042.39,E2 -1042.39} C_VEL
LIN {X 0,Y 594.376,Z 425.075,A -85,B 0,C 180,E1 -1044.671,E2 -1044.671} C_VEL
LIN {X 0,Y 594.373,Z 425.07,A -85,B 0,C 180,E1 -1047.087,E2 -1047.087} C_VEL
LIN {X 0,Y 594.392,Z 425.069,A -85,B 0,C 180,E1 -1049.668,E2 -1049.668} C_VEL
LIN {X 0,Y 594.364,Z 425.07,A -85,B 0,C 180,E1 -1052.538,E2 -1052.538} C_VEL
LIN {X 0,Y 594.371,Z 425.072,A -85,B 0,C 180,E1 -1054.807,E2 -1054.807} C_VEL
LIN {X 0,Y 594.396,Z 425.068,A -85,B 0,C 180,E1 -1057.254,E2 -1057.254} C_VEL
LIN {X 0,Y 594.373,Z 425.071,A -85,B 0,C 180,E1 -1059.946,E2 -1059.946} C_VEL
LIN {X 0,Y 594.387,Z 425.067,A -85,B 0,C 180,E1 -1062.806,E2 -1062.806} C_VEL
LIN {X 0,Y 594.379,Z 425.072,A -85,B 0,C 180,E1 -1065.825,E2 -1065.825} C_VEL
LIN {X 0,Y 594.387,Z 425.067,A -85,B 0,C 180,E1 -1068.404,E2 -1068.404} C_VEL
LIN {X 0,Y 594.399,Z 425.068,A -85,B 0,C 180,E1 -1071.158,E2 -1071.158} C_VEL
LIN {X 0,Y 594.39,Z 425.07,A -85,B 0,C 180,E1 -1073.891,E2 -1073.891} C_VEL
LIN {X 0,Y 594.381,Z 425.068,A -85,B 0,C 180,E1 -1076.611,E2 -1076.611} C_VEL
LIN {X 0,Y 594.417,Z 425.069,A -85,B 0,C 180,E1 -1079.322,E2 -1079.322} C_VEL
LIN {X 0,Y 594.388,Z 425.066,A -85,B 0,C 180,E1 -1082.033,E2 -1082.033} C_VEL
LIN {X 0,Y 594.396,Z 425.072,A -85,B 0,C 180,E1 -1084.748,E2 -1084.748} C_VEL
LIN {X 0,Y 594.411,Z 425.065,A -85,B 0,C 180,E1 -1087.473,E2 -1087.473} C_VEL
LIN {X 0,Y 594.397,Z 425.067,A -85,B 0,C 180,E1 -1090.216,E2 -1090.216} C_VEL
LIN {X 0,Y 594.366,Z 425.073,A -85,B 0,C 180,E1 -1092.983,E2 -1092.983} C_VEL
LIN {X 0,Y 594.368,Z 425.069,A -85,B 0,C 180,E1 -1095.781,E2 -1095.781} C_VEL
LIN {X 0,Y 594.382,Z 425.074,A -85,B 0,C 180,E1 -1098.618,E2 -1098.618} C_VEL
LIN {X 0,Y 594.365,Z 425.072,A -85,B 0,C 180,E1 -1101.503,E2 -1101.503} C_VEL
LIN {X 0,Y 594.379,Z 425.068,A -85,B 0,C 180,E1 -1104.447,E2 -1104.447} C_VEL
LIN {X 0,Y 594.384,Z 425.069,A -85,B 0,C 180,E1 -1106.7,E2 -1106.7} C_VEL
LIN {X 0,Y 594.378,Z 425.075,A -85,B 0,C 180,E1 -1108.999,E2 -1108.999} C_VEL
LIN {X 0,Y 594.387,Z 425.067,A -85,B 0,C 180,E1 -1111.647,E2 -1111.647} C_VEL
LIN {X 0,Y 594.388,Z 425.069,A -85,B 0,C 180,E1 -1114.579,E2 -1114.579} C_VEL
LIN {X 0,Y 594.379,Z 425.07,A -85,B 0,C 180,E1 -1117.087,E2 -1117.087} C_VEL
LIN {X 0,Y 594.369,Z 425.071,A -85,B 0,C 180,E1 -1119.775,E2 -1119.775} C_VEL
LIN {X 0,Y 594.383,Z 425.07,A -85,B 0,C 180,E1 -1122.374,E2 -1122.374} C_VEL
LIN {X 0,Y 594.356,Z 425.071,A -85,B 0,C 180,E1 -1125.192,E2 -1125.192} C_VEL
LIN {X 0,Y 594.383,Z 425.073,A -85,B 0,C 180,E1 -1128.152,E2 -1128.152} C_VEL
LIN {X 0,Y 594.39,Z 425.068,A -85,B 0,C 180,E1 -1130.322,E2 -1130.322} C_VEL
LIN {X 0,Y 594.381,Z 425.073,A -85,B 0,C 180,E1 -1132.914,E2 -1132.914} C_VEL
LIN {X 0,Y 594.382,Z 425.069,A -85,B 0,C 180,E1 -1135.861,E2 -1135.861} C_VEL
LIN {X 0,Y 594.4,Z 425.17,A -85,B 0,C 180,E1 -1137.364,E2 -1137.364} C_VEL
LIN {X 0,Y 594.704,Z 428.735,A -85,B 0,C 180,E1 -1138.307,E2 -1138.307} C_VEL
LIN {X 0,Y 594.634,Z 439.523,A -85,B 0,C 180,E1 -1141.016,E2 -1141.016} C_VEL
LIN {X 0,Y 594.539,Z 451.526,A -85,B 0,C 180,E1 -1143.947,E2 -1143.947} C_VEL
LIN {X 0,Y 594.514,Z 462.94,A -85,B 0,C 180,E1 -1146.672,E2 -1146.672} C_VEL
LIN {X 0,Y 594.445,Z 475.428,A -85,B 0,C 180,E1 -1149.589,E2 -1149.589} C_VEL
LIN {X 0,Y 594.4,Z 487.917,A -85,B 0,C 180,E1 -1152.453,E2 -1152.453} C_VEL
LIN {X 0,Y 594.351,Z 500.225,A -85,B 0,C 180,E1 -1155.233,E2 -1155.233} C_VEL
LIN {X 0,Y 594.349,Z 501.096,A -85,B 0,C 180,E1 -1155.428,E2 -1155.428} C_VEL
LIN {X 0,Y 594.881,Z 505.49,A -85,B 0,C 180,E1 -1155.502,E2 -1155.502} C_VEL
LIN {X 0,Y 594.84,Z 520.088,A -85,B 0,C 180,E1 -1155.784,E2 -1155.784} C_VEL
LIN {X 0,Y 594.756,Z 534.158,A -85,B 0,C 180,E1 -1156.2,E2 -1156.2} C_VEL
LIN {X 0,Y 594.686,Z 548.116,A -85,B 0,C 180,E1 -1156.764,E2 -1156.764} C_VEL
LIN {X 0,Y 594.603,Z 561.28,A -85,B 0,C 180,E1 -1157.457,E2 -1157.457} C_VEL
LIN {X 0,Y 594.533,Z 573.163,A -85,B 0,C 180,E1 -1158.235,E2 -1158.235} C_VEL
LIN {X 0,Y 594.475,Z 584.004,A -85,B 0,C 180,E1 -1159.097,E2 -1159.097} C_VEL
LIN {X 0,Y 594.375,Z 594.717,A -85,B 0,C 180,E1 -1160.129,E2 -1160.129} C_VEL
LIN {X 0,Y 594.351,Z 603.566,A -85,B 0,C 180,E1 -1161.158,E2 -1161.158} C_VEL
LIN {X 0,Y 594.315,Z 612.045,A -85,B 0,C 180,E1 -1162.356,E2 -1162.356} C_VEL
LIN {X 0,Y 594.27,Z 619.233,A -85,B 0,C 180,E1 -1163.619,E2 -1163.619} C_VEL
LIN {X 0,Y 594.248,Z 624.965,A -85,B 0,C 180,E1 -1164.912,E2 -1164.912} C_VEL
LIN {X 0,Y 594.259,Z 628.444,A -85,B 0,C 180,E1 -1165.932,E2 -1165.932} C_VEL
LIN {X 0,Y 594.224,Z 631.833,A -85,B 0,C 180,E1 -1167.289,E2 -1167.289} C_VEL
LIN {X 0,Y 594.242,Z 633.832,A -85,B 0,C 180,E1 -1168.645,E2 -1168.645} C_VEL
LIN {X 0,Y 594.234,Z 634.5,A -85,B 0,C 180,E1 -1170.001,E2 -1170.001} C_VEL
LIN {X 0,Y 594.242,Z 633.83,A -85,B 0,C 180,E1 -1171.356,E2 -1171.356} C_VEL
LIN {X 0,Y 594.224,Z 631.83,A -85,B 0,C 180,E1 -1172.712,E2 -1172.712} C_VEL
LIN {X 0,Y 594.259,Z 628.44,A -85,B 0,C 180,E1 -1174.07,E2 -1174.07} C_VEL
LIN {X 0,Y 594.275,Z 623.564,A -85,B 0,C 180,E1 -1175.43,E2 -1175.43} C_VEL
LIN {X 0,Y 594.3,Z 618.031,A -85,B 0,C 180,E1 -1176.607,E2 -1176.607} C_VEL
LIN {X 0,Y 594.316,Z 610.914,A -85,B 0,C 180,E1 -1177.817,E2 -1177.817} C_VEL
LIN {X 0,Y 594.369,Z 602.192,A -85,B 0,C 180,E1 -1179.015,E2 -1179.015} C_VEL
LIN {X 0,Y 594.4,Z 593.074,A -85,B 0,C 180,E1 -1180.044,E2 -1180.044} C_VEL
LIN {X 0,Y 594.48,Z 582.695,A -85,B 0,C 180,E1 -1181.018,E2 -1181.018} C_VEL
LIN {X 0,Y 594.576,Z 570.693,A -85,B 0,C 180,E1 -1181.939,E2 -1181.939} C_VEL
LIN {X 0,Y 594.605,Z 558.197,A -85,B 0,C 180,E1 -1182.718,E2 -1182.718} C_VEL
LIN {X 0,Y 594.687,Z 546.111,A -85,B 0,C 180,E1 -1183.324,E2 -1183.324} C_VEL
LIN {X 0,Y 594.779,Z 532.178,A -85,B 0,C 180,E1 -1183.866,E2 -1183.866} C_VEL
LIN {X 0,Y 594.842,Z 518.26,A -85,B 0,C 180,E1 -1184.259,E2 -1184.259} C_VEL
LIN {X 0,Y 594.838,Z 503.907,A -85,B 0,C 180,E1 -1184.522,E2 -1184.522} C_VEL
LIN {X 0,Y 594.355,Z 501.079,A -85,B 0,C 180,E1 -1184.576,E2 -1184.576} C_VEL
LIN {X 0,Y 594.411,Z 489.47,A -85,B 0,C 180,E1 -1187.193,E2 -1187.193} C_VEL
LIN {X 0,Y 594.45,Z 476.981,A -85,B 0,C 180,E1 -1190.052,E2 -1190.052} C_VEL
LIN {X 0,Y 594.498,Z 464.493,A -85,B 0,C 180,E1 -1192.962,E2 -1192.962} C_VEL
LIN {X 0,Y 594.548,Z 453.565,A -85,B 0,C 180,E1 -1195.561,E2 -1195.561} C_VEL
LIN {X 0,Y 594.617,Z 442.638,A -85,B 0,C 180,E1 -1198.215,E2 -1198.215} C_VEL
LIN {X 0,Y 594.68,Z 431.71,A -85,B 0,C 180,E1 -1200.937,E2 -1200.937} C_VEL
LIN {X 0,Y 594.739,Z 427.145,A -85,B 0,C 180,E1 -1202.125,E2 -1202.125} C_VEL
LIN {X 0,Y 594.395,Z 425.074,A -85,B 0,C 180,E1 -1202.789,E2 -1202.789} C_VEL
LIN {X 0,Y 594.363,Z 425.074,A -85,B 0,C 180,E1 -1205.409,E2 -1205.409} C_VEL
LIN {X 0,Y 594.389,Z 425.071,A -85,B 0,C 180,E1 -1207.941,E2 -1207.941} C_VEL
LIN {X 0,Y 594.378,Z 425.073,A -85,B 0,C 180,E1 -1210.822,E2 -1210.822} C_VEL
LIN {X 0,Y 594.371,Z 425.077,A -85,B 0,C 180,E1 -1213.3,E2 -1213.3} C_VEL
LIN {X 0,Y 594.388,Z 425.074,A -85,B 0,C 180,E1 -1216.159,E2 -1216.159} C_VEL
LIN {X 0,Y 594.381,Z 425.076,A -85,B 0,C 180,E1 -1219.178,E2 -1219.178} C_VEL
LIN {X 0,Y 594.389,Z 425.074,A -85,B 0,C 180,E1 -1222.059,E2 -1222.059} C_VEL
LIN {X 0,Y 594.433,Z 425.268,A -85,B 0,C 180,E1 -1224.861,E2 -1224.861} C_VEL
LIN {X 0,Y 594.371,Z 432.03,A -85,B 0,C 180,E1 -1227.853,E2 -1227.853} C_VEL
LIN {X 0,Y 594.367,Z 437.32,A -85,B 0,C 180,E1 -1230.223,E2 -1230.223} C_VEL
LIN {X 0,Y 594.339,Z 442.418,A -85,B 0,C 180,E1 -1232.537,E2 -1232.537} C_VEL
LIN {X 0,Y 594.345,Z 449.282,A -85,B 0,C 180,E1 -1235.552,E2 -1235.552} C_VEL
LIN {X 0,Y 594.29,Z 456.146,A -85,B 0,C 180,E1 -1238.494,E2 -1238.494} C_VEL
LIN {X 0,Y 594.289,Z 463.01,A -85,B 0,C 180,E1 -1241.379,E2 -1241.379} C_VEL
LIN {X 0,Y 594.263,Z 469.875,A -85,B 0,C 180,E1 -1244.216,E2 -1244.216} C_VEL
LIN {X 0,Y 594.257,Z 475.024,A -85,B 0,C 180,E1 -1246.318,E2 -1246.318} C_VEL
LIN {X 0,Y 594.265,Z 479.207,A -85,B 0,C 180,E1 -1248.012,E2 -1248.012} C_VEL
LIN {X 0,Y 594.673,Z 483.78,A -85,B 0,C 180,E1 -1248.107,E2 -1248.107} C_VEL
LIN {X 0,Y 594.618,Z 495.932,A -85,B 0,C 180,E1 -1248.409,E2 -1248.409} C_VEL
LIN {X 0,Y 594.56,Z 508.106,A -85,B 0,C 180,E1 -1248.845,E2 -1248.845} C_VEL
LIN {X 0,Y 594.509,Z 520.458,A -85,B 0,C 180,E1 -1249.442,E2 -1249.442} C_VEL
LIN {X 0,Y 594.448,Z 531.586,A -85,B 0,C 180,E1 -1250.129,E2 -1250.129} C_VEL
LIN {X 0,Y 594.406,Z 540.6,A -85,B 0,C 180,E1 -1250.815,E2 -1250.815} C_VEL
LIN {X 0,Y 594.373,Z 549.86,A -85,B 0,C 180,E1 -1251.672,E2 -1251.672} C_VEL
LIN {X 0,Y 594.317,Z 558.833,A -85,B 0,C 180,E1 -1252.697,E2 -1252.697} C_VEL
LIN {X 0,Y 594.285,Z 565.358,A -85,B 0,C 180,E1 -1253.612,E2 -1253.612} C_VEL
LIN {X 0,Y 594.289,Z 570.941,A -85,B 0,C 180,E1 -1254.571,E2 -1254.571} C_VEL
LIN {X 0,Y 594.27,Z 575.683,A -85,B 0,C 180,E1 -1255.591,E2 -1255.591} C_VEL
LIN {X 0,Y 594.268,Z 579.317,A -85,B 0,C 180,E1 -1256.61,E2 -1256.61} C_VEL
LIN {X 0,Y 594.225,Z 581.194,A -85,B 0,C 180,E1 -1257.288,E2 -1257.288} C_VEL
LIN {X 0,Y 594.24,Z 582.627,A -85,B 0,C 180,E1 -1257.967,E2 -1257.967} C_VEL
LIN {X 0,Y 594.24,Z 584.253,A -85,B 0,C 180,E1 -1259.322,E2 -1259.322} C_VEL
LIN {X 0,Y 594.236,Z 584.496,A -85,B 0,C 180,E1 -1260,E2 -1260} C_VEL
LIN {X 0,Y 594.24,Z 584.315,A -85,B 0,C 180,E1 -1260.678,E2 -1260.678} C_VEL
LIN {X 0,Y 594.239,Z 582.775,A -85,B 0,C 180,E1 -1262.033,E2 -1262.033} C_VEL
LIN {X 0,Y 594.226,Z 581.415,A -85,B 0,C 180,E1 -1262.712,E2 -1262.712} C_VEL
LIN {X 0,Y 594.289,Z 578.538,A -85,B 0,C 180,E1 -1263.729,E2 -1263.729} C_VEL
LIN {X 0,Y 594.242,Z 574.638,A -85,B 0,C 180,E1 -1264.749,E2 -1264.749} C_VEL
LIN {X 0,Y 594.299,Z 569.606,A -85,B 0,C 180,E1 -1265.769,E2 -1265.769} C_VEL
LIN {X 0,Y 594.317,Z 563.287,A -85,B 0,C 180,E1 -1266.791,E2 -1266.791} C_VEL
LIN {X 0,Y 594.347,Z 555.369,A -85,B 0,C 180,E1 -1267.816,E2 -1267.816} C_VEL
LIN {X 0,Y 594.381,Z 545.523,A -85,B 0,C 180,E1 -1268.842,E2 -1268.842} C_VEL
LIN {X 0,Y 594.427,Z 535.201,A -85,B 0,C 180,E1 -1269.7,E2 -1269.7} C_VEL
LIN {X 0,Y 594.502,Z 523.578,A -85,B 0,C 180,E1 -1270.472,E2 -1270.472} C_VEL
LIN {X 0,Y 594.56,Z 511.795,A -85,B 0,C 180,E1 -1271.084,E2 -1271.084} C_VEL
LIN {X 0,Y 594.59,Z 499.995,A -85,B 0,C 180,E1 -1271.55,E2 -1271.55} C_VEL
LIN {X 0,Y 594.657,Z 491.228,A -85,B 0,C 180,E1 -1271.814,E2 -1271.814} C_VEL
LIN {X 0,Y 593.904,Z 487.394,A -85,B 0,C 180,E1 -1271.952,E2 -1271.952} C_VEL
LIN {X 0,Y 591.57,Z 483.063,A -85,B 0,C 180,E1 -1272.219,E2 -1272.219} C_VEL
LIN {X 0,Y 588.961,Z 479.669,A -85,B 0,C 180,E1 -1272.575,E2 -1272.575} C_VEL
LIN {X 0,Y 587.528,Z 477.775,A -85,B 0,C 180,E1 -1272.908,E2 -1272.908} C_VEL
LIN {X 0,Y 587.175,Z 476.924,A -85,B 0,C 180,E1 -1273.16,E2 -1273.16} C_VEL
LIN {X 0,Y 587.183,Z 471.81,A -85,B 0,C 180,E1 -1275.267,E2 -1275.267} C_VEL
LIN {X 0,Y 587.214,Z 466.659,A -85,B 0,C 180,E1 -1277.41,E2 -1277.41} C_VEL
LIN {X 0,Y 587.217,Z 461.508,A -85,B 0,C 180,E1 -1279.58,E2 -1279.58} C_VEL
LIN {X 0,Y 587.265,Z 454.639,A -85,B 0,C 180,E1 -1282.517,E2 -1282.517} C_VEL
LIN {X 0,Y 587.259,Z 447.771,A -85,B 0,C 180,E1 -1285.52,E2 -1285.52} C_VEL
LIN {X 0,Y 587.271,Z 442.619,A -85,B 0,C 180,E1 -1287.822,E2 -1287.822} C_VEL
LIN {X 0,Y 587.318,Z 437.487,A -85,B 0,C 180,E1 -1290.171,E2 -1290.171} C_VEL
LIN {X 0,Y 587.343,Z 432.3,A -85,B 0,C 180,E1 -1292.579,E2 -1292.579} C_VEL
LIN {X 0,Y 587.364,Z 427.05,A -85,B 0,C 180,E1 -1295.053,E2 -1295.053} C_VEL
LIN {X 0,Y 587.344,Z 425.951,A -85,B 0,C 180,E1 -1295.691,E2 -1295.691} C_VEL
LIN {X 0,Y 587.327,Z 425.954,A -85,B 0,C 180,E1 -1298.48,E2 -1298.48} C_VEL
LIN {X 0,Y 587.341,Z 425.95,A -85,B 0,C 180,E1 -1301.157,E2 -1301.157} C_VEL
LIN {X 0,Y 587.34,Z 425.951,A -85,B 0,C 180,E1 -1304.114,E2 -1304.114} C_VEL
LIN {X 0,Y 587.316,Z 425.955,A -85,B 0,C 180,E1 -1306.993,E2 -1306.993} C_VEL
LIN {X 0,Y 587.321,Z 425.953,A -85,B 0,C 180,E1 -1309.746,E2 -1309.746} C_VEL
LIN {X 0,Y 587.39,Z 426.094,A -85,B 0,C 180,E1 -1312.156,E2 -1312.156} C_VEL
LIN {X 0,Y 587.373,Z 434.304,A -85,B 0,C 180,E1 -1314.947,E2 -1314.947} C_VEL
LIN {X 0,Y 587.377,Z 442.68,A -85,B 0,C 180,E1 -1317.821,E2 -1317.821} C_VEL
LIN {X 0,Y 587.459,Z 450.808,A -85,B 0,C 180,E1 -1320.626,E2 -1320.626} C_VEL
LIN {X 0,Y 587.371,Z 459.624,A -85,B 0,C 180,E1 -1323.817,E2 -1323.817} C_VEL
LIN {X 0,Y 587.344,Z 466.839,A -85,B 0,C 180,E1 -1326.368,E2 -1326.368} C_VEL
LIN {X 0,Y 587.294,Z 475.404,A -85,B 0,C 180,E1 -1329.332,E2 -1329.332} C_VEL
LIN {X 0,Y 587.256,Z 483.94,A -85,B 0,C 180,E1 -1332.231,E2 -1332.231} C_VEL
LIN {X 0,Y 587.216,Z 492.491,A -85,B 0,C 180,E1 -1335.088,E2 -1335.088} C_VEL
LIN {X 0,Y 587.235,Z 493.269,A -85,B 0,C 180,E1 -1335.321,E2 -1335.321} C_VEL
LIN {X 0,Y 588.007,Z 498.387,A -85,B 0,C 180,E1 -1335.419,E2 -1335.419} C_VEL
LIN {X 0,Y 587.938,Z 512.895,A -85,B 0,C 180,E1 -1335.728,E2 -1335.728} C_VEL
LIN {X 0,Y 587.828,Z 527.638,A -85,B 0,C 180,E1 -1336.209,E2 -1336.209} C_VEL
LIN {X 0,Y 587.743,Z 540.717,A -85,B 0,C 180,E1 -1336.779,E2 -1336.779} C_VEL
LIN {X 0,Y 587.619,Z 553.37,A -85,B 0,C 180,E1 -1337.479,E2 -1337.479} C_VEL
LIN {X 0,Y 587.515,Z 566.037,A -85,B 0,C 180,E1 -1338.353,E2 -1338.353} C_VEL
LIN {X 0,Y 587.467,Z 575.421,A -85,B 0,C 180,E1 -1339.139,E2 -1339.139} C_VEL
LIN {X 0,Y 587.355,Z 585.885,A -85,B 0,C 180,E1 -1340.182,E2 -1340.182} C_VEL
LIN {X 0,Y 587.311,Z 594.555,A -85,B 0,C 180,E1 -1341.223,E2 -1341.223} C_VEL
LIN {X 0,Y 587.25,Z 602.83,A -85,B 0,C 180,E1 -1342.435,E2 -1342.435} C_VEL
LIN {X 0,Y 587.18,Z 609.451,A -85,B 0,C 180,E1 -1343.636,E2 -1343.636} C_VEL
LIN {X 0,Y 587.159,Z 614.773,A -85,B 0,C 180,E1 -1344.849,E2 -1344.849} C_VEL
LIN {X 0,Y 587.181,Z 618.293,A -85,B 0,C 180,E1 -1345.881,E2 -1345.881} C_VEL
LIN {X 0,Y 587.13,Z 621.74,A -85,B 0,C 180,E1 -1347.255,E2 -1347.255} C_VEL
LIN {X 0,Y 587.145,Z 623.786,A -85,B 0,C 180,E1 -1348.627,E2 -1348.627} C_VEL
LIN {X 0,Y 587.136,Z 624.48,A -85,B 0,C 180,E1 -1349.999,E2 -1349.999} C_VEL
LIN {X 0,Y 587.142,Z 623.874,A -85,B 0,C 180,E1 -1351.371,E2 -1351.371} C_VEL
LIN {X 0,Y 587.128,Z 621.931,A -85,B 0,C 180,E1 -1352.744,E2 -1352.744} C_VEL
LIN {X 0,Y 587.182,Z 618.576,A -85,B 0,C 180,E1 -1354.117,E2 -1354.117} C_VEL
LIN {X 0,Y 587.2,Z 613.755,A -85,B 0,C 180,E1 -1355.494,E2 -1355.494} C_VEL
LIN {X 0,Y 587.209,Z 607.301,A -85,B 0,C 180,E1 -1356.873,E2 -1356.873} C_VEL
LIN {X 0,Y 587.268,Z 600.103,A -85,B 0,C 180,E1 -1358.083,E2 -1358.083} C_VEL
LIN {X 0,Y 587.332,Z 592.555,A -85,B 0,C 180,E1 -1359.122,E2 -1359.122} C_VEL
LIN {X 0,Y 587.375,Z 583.492,A -85,B 0,C 180,E1 -1360.164,E2 -1360.164} C_VEL
LIN {X 0,Y 587.464,Z 574.502,A -85,B 0,C 180,E1 -1361.034,E2 -1361.034} C_VEL
LIN {X 0,Y 587.569,Z 562.604,A -85,B 0,C 180,E1 -1361.994,E2 -1361.994} C_VEL
LIN {X 0,Y 587.637,Z 550.532,A -85,B 0,C 180,E1 -1362.782,E2 -1362.782} C_VEL
LIN {X 0,Y 587.765,Z 538.997,A -85,B 0,C 180,E1 -1363.394,E2 -1363.394} C_VEL
LIN {X 0,Y 587.847,Z 525.701,A -85,B 0,C 180,E1 -1363.957,E2 -1363.957} C_VEL
LIN {X 0,Y 587.937,Z 511.302,A -85,B 0,C 180,E1 -1364.401,E2 -1364.401} C_VEL
LIN {X 0,Y 587.94,Z 496.969,A -85,B 0,C 180,E1 -1364.696,E2 -1364.696} C_VEL
LIN {X 0,Y 587.218,Z 493.169,A -85,B 0,C 180,E1 -1364.777,E2 -1364.777} C_VEL
LIN {X 0,Y 587.247,Z 485.282,A -85,B 0,C 180,E1 -1367.408,E2 -1367.408} C_VEL
LIN {X 0,Y 587.282,Z 476.727,A -85,B 0,C 180,E1 -1370.305,E2 -1370.305} C_VEL
LIN {X 0,Y 587.326,Z 468.171,A -85,B 0,C 180,E1 -1373.257,E2 -1373.257} C_VEL
LIN {X 0,Y 587.374,Z 461.754,A -85,B 0,C 180,E1 -1375.514,E2 -1375.514} C_VEL
LIN {X 0,Y 587.408,Z 454.267,A -85,B 0,C 180,E1 -1378.202,E2 -1378.202} C_VEL
LIN {X 0,Y 587.421,Z 447.792,A -85,B 0,C 180,E1 -1380.523,E2 -1380.523} C_VEL
LIN {X 0,Y 587.378,Z 439.43,A -85,B 0,C 180,E1 -1383.392,E2 -1383.392} C_VEL
LIN {X 0,Y 587.396,Z 430.933,A -85,B 0,C 180,E1 -1386.302,E2 -1386.302} C_VEL
LIN {X 0,Y 587.361,Z 425.946,A -85,B 0,C 180,E1 -1388.045,E2 -1388.045} C_VEL
LIN {X 0,Y 587.333,Z 425.952,A -85,B 0,C 180,E1 -1391.074,E2 -1391.074} C_VEL
LIN {X 0,Y 587.328,Z 425.951,A -85,B 0,C 180,E1 -1394.113,E2 -1394.113} C_VEL
LIN {X 0,Y 587.33,Z 425.947,A -85,B 0,C 180,E1 -1396.995,E2 -1396.995} C_VEL
LIN {X 0,Y 587.314,Z 425.954,A -85,B 0,C 180,E1 -1399.745,E2 -1399.745} C_VEL
LIN {X 0,Y 587.34,Z 425.945,A -85,B 0,C 180,E1 -1402.392,E2 -1402.392} C_VEL
LIN {X 0,Y 587.342,Z 425.95,A -85,B 0,C 180,E1 -1404.945,E2 -1404.945} C_VEL
LIN {X 0,Y 587.335,Z 425.946,A -85,B 0,C 180,E1 -1407.421,E2 -1407.421} C_VEL
LIN {X 0,Y 587.339,Z 425.95,A -85,B 0,C 180,E1 -1409.83,E2 -1409.83} C_VEL
LIN {X 0,Y 587.342,Z 425.945,A -85,B 0,C 180,E1 -1412.306,E2 -1412.306} C_VEL
LIN {X 0,Y 587.33,Z 425.946,A -85,B 0,C 180,E1 -1414.483,E2 -1414.483} C_VEL
LIN {X 0,Y 587.361,Z 425.942,A -85,B 0,C 180,E1 -1417.487,E2 -1417.487} C_VEL
LIN {X 0,Y 587.338,Z 425.953,A -85,B 0,C 180,E1 -1420.425,E2 -1420.425} C_VEL
LIN {X 0,Y 587.349,Z 425.945,A -85,B 0,C 180,E1 -1423.311,E2 -1423.311} C_VEL
LIN {X 0,Y 587.351,Z 425.944,A -85,B 0,C 180,E1 -1426.154,E2 -1426.154} C_VEL
LIN {X 0,Y 587.341,Z 425.951,A -85,B 0,C 180,E1 -1428.962,E2 -1428.962} C_VEL
LIN {X 0,Y 587.364,Z 425.942,A -85,B 0,C 180,E1 -1431.745,E2 -1431.745} C_VEL
LIN {X 0,Y 587.361,Z 425.946,A -85,B 0,C 180,E1 -1434.507,E2 -1434.507} C_VEL
LIN {X 0,Y 587.373,Z 425.943,A -85,B 0,C 180,E1 -1437.257,E2 -1437.257} C_VEL
LIN {X 0,Y 587.373,Z 425.942,A -85,B 0,C 180,E1 -1440,E2 -1440} C_VEL
LIN {X 0,Y 587.376,Z 425.945,A -85,B 0,C 180,E1 -1442.743,E2 -1442.743} C_VEL
LIN {X 0,Y 587.355,Z 425.943,A -85,B 0,C 180,E1 -1445.493,E2 -1445.493} C_VEL
LIN {X 0,Y 587.366,Z 425.947,A -85,B 0,C 180,E1 -1448.255,E2 -1448.255} C_VEL
LIN {X 0,Y 587.351,Z 425.944,A -85,B 0,C 180,E1 -1451.142,E2 -1451.142} C_VEL
LIN {X 0,Y 587.354,Z 425.943,A -85,B 0,C 180,E1 -1454.261,E2 -1454.261} C_VEL
LIN {X 0,Y 587.352,Z 425.942,A -85,B 0,C 180,E1 -1457.406,E2 -1457.406} C_VEL
LIN {X 0,Y 587.328,Z 425.953,A -85,B 0,C 180,E1 -1460.305,E2 -1460.305} C_VEL
LIN {X 0,Y 587.317,Z 425.95,A -85,B 0,C 180,E1 -1463.259,E2 -1463.259} C_VEL
LIN {X 0,Y 587.353,Z 425.943,A -85,B 0,C 180,E1 -1466.183,E2 -1466.183} C_VEL
LIN {X 0,Y 587.345,Z 425.949,A -85,B 0,C 180,E1 -1469.135,E2 -1469.135} C_VEL
LIN {X 0,Y 587.351,Z 425.945,A -85,B 0,C 180,E1 -1471.839,E2 -1471.839} C_VEL
LIN {X 0,Y 587.35,Z 425.948,A -85,B 0,C 180,E1 -1474.35,E2 -1474.35} C_VEL
LIN {X 0,Y 587.345,Z 425.944,A -85,B 0,C 180,E1 -1476.747,E2 -1476.747} C_VEL
LIN {X 0,Y 587.338,Z 425.952,A -85,B 0,C 180,E1 -1479.36,E2 -1479.36} C_VEL
LIN {X 0,Y 587.359,Z 425.943,A -85,B 0,C 180,E1 -1482.112,E2 -1482.112} C_VEL
LIN {X 0,Y 587.308,Z 425.95,A -85,B 0,C 180,E1 -1485.09,E2 -1485.09} C_VEL
LIN {X 0,Y 587.346,Z 425.952,A -85,B 0,C 180,E1 -1487.929,E2 -1487.929} C_VEL
LIN {X 0,Y 587.343,Z 425.945,A -85,B 0,C 180,E1 -1490.642,E2 -1490.642} C_VEL
LIN {X 0,Y 587.349,Z 425.951,A -85,B 0,C 180,E1 -1493.293,E2 -1493.293} C_VEL
LIN {X 0,Y 587.366,Z 425.944,A -85,B 0,C 180,E1 -1495.782,E2 -1495.782} C_VEL
LIN {X 0,Y 587.359,Z 426.123,A -85,B 0,C 180,E1 -1497.155,E2 -1497.155} C_VEL
LIN {X 0,Y 587.799,Z 429.539,A -85,B 0,C 180,E1 -1498.093,E2 -1498.093} C_VEL
LIN {X 0,Y 587.661,Z 441.419,A -85,B 0,C 180,E1 -1501.115,E2 -1501.115} C_VEL
LIN {X 0,Y 587.572,Z 452.189,A -85,B 0,C 180,E1 -1503.777,E2 -1503.777} C_VEL
LIN {X 0,Y 587.507,Z 462.94,A -85,B 0,C 180,E1 -1506.377,E2 -1506.377} C_VEL
LIN {X 0,Y 587.412,Z 473.867,A -85,B 0,C 180,E1 -1508.967,E2 -1508.967} C_VEL
LIN {X 0,Y 587.392,Z 486.356,A -85,B 0,C 180,E1 -1511.877,E2 -1511.877} C_VEL
LIN {X 0,Y 587.316,Z 498.844,A -85,B 0,C 180,E1 -1514.738,E2 -1514.738} C_VEL
LIN {X 0,Y 587.296,Z 501.089,A -85,B 0,C 180,E1 -1515.247,E2 -1515.247} C_VEL
LIN {X 0,Y 588.022,Z 505.695,A -85,B 0,C 180,E1 -1515.332,E2 -1515.332} C_VEL
LIN {X 0,Y 587.939,Z 519.839,A -85,B 0,C 180,E1 -1515.608,E2 -1515.608} C_VEL
LIN {X 0,Y 587.884,Z 532.579,A -85,B 0,C 180,E1 -1515.981,E2 -1515.981} C_VEL
LIN {X 0,Y 587.774,Z 546.153,A -85,B 0,C 180,E1 -1516.518,E2 -1516.518} C_VEL
LIN {X 0,Y 587.638,Z 558.23,A -85,B 0,C 180,E1 -1517.13,E2 -1517.13} C_VEL
LIN {X 0,Y 587.587,Z 570.72,A -85,B 0,C 180,E1 -1517.919,E2 -1517.919} C_VEL
LIN {X 0,Y 587.459,Z 582.281,A -85,B 0,C 180,E1 -1518.813,E2 -1518.813} C_VEL
LIN {X 0,Y 587.376,Z 593.09,A -85,B 0,C 180,E1 -1519.836,E2 -1519.836} C_VEL
LIN {X 0,Y 587.338,Z 602.207,A -85,B 0,C 180,E1 -1520.878,E2 -1520.878} C_VEL
LIN {X 0,Y 587.26,Z 610.926,A -85,B 0,C 180,E1 -1522.09,E2 -1522.09} C_VEL
LIN {X 0,Y 587.208,Z 618.527,A -85,B 0,C 180,E1 -1523.407,E2 -1523.407} C_VEL
LIN {X 0,Y 587.199,Z 623.572,A -85,B 0,C 180,E1 -1524.506,E2 -1524.506} C_VEL
LIN {X 0,Y 587.179,Z 628.445,A -85,B 0,C 180,E1 -1525.883,E2 -1525.883} C_VEL
LIN {X 0,Y 587.13,Z 631.833,A -85,B 0,C 180,E1 -1527.257,E2 -1527.257} C_VEL
LIN {X 0,Y 587.141,Z 633.832,A -85,B 0,C 180,E1 -1528.629,E2 -1528.629} C_VEL
LIN {X 0,Y 587.135,Z 634.5,A -85,B 0,C 180,E1 -1530.001,E2 -1530.001} C_VEL
LIN {X 0,Y 587.141,Z 633.831,A -85,B 0,C 180,E1 -1531.373,E2 -1531.373} C_VEL
LIN {X 0,Y 587.13,Z 631.831,A -85,B 0,C 180,E1 -1532.745,E2 -1532.745} C_VEL
LIN {X 0,Y 587.179,Z 628.44,A -85,B 0,C 180,E1 -1534.119,E2 -1534.119} C_VEL
LIN {X 0,Y 587.199,Z 623.564,A -85,B 0,C 180,E1 -1535.495,E2 -1535.495} C_VEL
LIN {X 0,Y 587.21,Z 617.048,A -85,B 0,C 180,E1 -1536.875,E2 -1536.875} C_VEL
LIN {X 0,Y 587.269,Z 609.794,A -85,B 0,C 180,E1 -1538.084,E2 -1538.084} C_VEL
LIN {X 0,Y 587.322,Z 600.816,A -85,B 0,C 180,E1 -1539.297,E2 -1539.297} C_VEL
LIN {X 0,Y 587.372,Z 591.383,A -85,B 0,C 180,E1 -1540.34,E2 -1540.34} C_VEL
LIN {X 0,Y 587.476,Z 581.019,A -85,B 0,C 180,E1 -1541.291,E2 -1541.291} C_VEL
LIN {X 0,Y 587.579,Z 569.418,A -85,B 0,C 180,E1 -1542.171,E2 -1542.171} C_VEL
LIN {X 0,Y 587.667,Z 556.633,A -85,B 0,C 180,E1 -1542.959,E2 -1542.959} C_VEL
LIN {X 0,Y 587.789,Z 544.143,A -85,B 0,C 180,E1 -1543.572,E2 -1543.572} C_VEL
LIN {X 0,Y 587.904,Z 530.71,A -85,B 0,C 180,E1 -1544.082,E2 -1544.082} C_VEL
LIN {X 0,Y 587.945,Z 516.967,A -85,B 0,C 180,E1 -1544.461,E2 -1544.461} C_VEL
LIN {X 0,Y 587.937,Z 504.55,A -85,B 0,C 180,E1 -1544.687,E2 -1544.687} C_VEL
LIN {X 0,Y 587.304,Z 500.983,A -85,B 0,C 180,E1 -1544.777,E2 -1544.777} C_VEL
LIN {X 0,Y 587.362,Z 487.909,A -85,B 0,C 180,E1 -1547.766,E2 -1547.766} C_VEL
LIN {X 0,Y 587.415,Z 475.42,A -85,B 0,C 180,E1 -1550.668,E2 -1550.668} C_VEL
LIN {X 0,Y 587.511,Z 464.493,A -85,B 0,C 180,E1 -1553.252,E2 -1553.252} C_VEL
LIN {X 0,Y 587.581,Z 453.655,A -85,B 0,C 180,E1 -1555.864,E2 -1555.864} C_VEL
LIN {X 0,Y 587.665,Z 442.638,A -85,B 0,C 180,E1 -1558.58,E2 -1558.58} C_VEL
LIN {X 0,Y 587.774,Z 433.381,A -85,B 0,C 180,E1 -1560.941,E2 -1560.941} C_VEL
LIN {X 0,Y 587.833,Z 428.74,A -85,B 0,C 180,E1 -1562.183,E2 -1562.183} C_VEL
LIN {X 0,Y 587.329,Z 425.954,A -85,B 0,C 180,E1 -1563.049,E2 -1563.049} C_VEL
LIN {X 0,Y 587.335,Z 425.95,A -85,B 0,C 180,E1 -1565.543,E2 -1565.543} C_VEL
LIN {X 0,Y 587.343,Z 425.95,A -85,B 0,C 180,E1 -1567.839,E2 -1567.839} C_VEL
LIN {X 0,Y 587.322,Z 425.954,A -85,B 0,C 180,E1 -1570.254,E2 -1570.254} C_VEL
LIN {X 0,Y 587.319,Z 425.953,A -85,B 0,C 180,E1 -1573.119,E2 -1573.119} C_VEL
LIN {X 0,Y 587.34,Z 425.951,A -85,B 0,C 180,E1 -1576.051,E2 -1576.051} C_VEL
LIN {X 0,Y 587.341,Z 425.95,A -85,B 0,C 180,E1 -1578.925,E2 -1578.925} C_VEL
LIN {X 0,Y 587.327,Z 425.95,A -85,B 0,C 180,E1 -1581.52,E2 -1581.52} C_VEL
LIN {X 0,Y 587.357,Z 425.948,A -85,B 0,C 180,E1 -1584.455,E2 -1584.455} C_VEL
LIN {X 0,Y 587.371,Z 426.093,A -85,B 0,C 180,E1 -1584.772,E2 -1584.772} C_VEL
LIN {X 0,Y 587.343,Z 431.989,A -85,B 0,C 180,E1 -1587.421,E2 -1587.421} C_VEL
LIN {X 0,Y 587.32,Z 437.32,A -85,B 0,C 180,E1 -1589.829,E2 -1589.829} C_VEL
LIN {X 0,Y 587.301,Z 442.725,A -85,B 0,C 180,E1 -1592.318,E2 -1592.318} C_VEL
LIN {X 0,Y 587.265,Z 449.284,A -85,B 0,C 180,E1 -1595.238,E2 -1595.238} C_VEL
LIN {X 0,Y 587.229,Z 456.148,A -85,B 0,C 180,E1 -1598.222,E2 -1598.222} C_VEL
LIN {X 0,Y 587.245,Z 463.012,A -85,B 0,C 180,E1 -1601.148,E2 -1601.148} C_VEL
LIN {X 0,Y 587.181,Z 469.877,A -85,B 0,C 180,E1 -1604.021,E2 -1604.021} C_VEL
LIN {X 0,Y 587.191,Z 475.025,A -85,B 0,C 180,E1 -1606.15,E2 -1606.15} C_VEL
LIN {X 0,Y 587.161,Z 479.209,A -85,B 0,C 180,E1 -1607.865,E2 -1607.865} C_VEL
LIN {X 0,Y 587.721,Z 484.947,A -85,B 0,C 180,E1 -1607.986,E2 -1607.986} C_VEL
LIN {X 0,Y 587.662,Z 497.419,A -85,B 0,C 180,E1 -1608.316,E2 -1608.316} C_VEL
LIN {X 0,Y 587.559,Z 509.943,A -85,B 0,C 180,E1 -1608.791,E2 -1608.791} C_VEL
LIN {X 0,Y 587.523,Z 522.036,A -85,B 0,C 180,E1 -1609.402,E2 -1609.402} C_VEL
LIN {X 0,Y 587.432,Z 532.823,A -85,B 0,C 180,E1 -1610.097,E2 -1610.097} C_VEL
LIN {X 0,Y 587.357,Z 542.598,A -85,B 0,C 180,E1 -1610.878,E2 -1610.878} C_VEL
LIN {X 0,Y 587.302,Z 551.491,A -85,B 0,C 180,E1 -1611.744,E2 -1611.744} C_VEL
LIN {X 0,Y 587.274,Z 560.176,A -85,B 0,C 180,E1 -1612.781,E2 -1612.781} C_VEL
LIN {X 0,Y 587.214,Z 567.104,A -85,B 0,C 180,E1 -1613.816,E2 -1613.816} C_VEL
LIN {X 0,Y 587.167,Z 572.654,A -85,B 0,C 180,E1 -1614.85,E2 -1614.85} C_VEL
LIN {X 0,Y 587.182,Z 577.016,A -85,B 0,C 180,E1 -1615.882,E2 -1615.882} C_VEL
LIN {X 0,Y 587.195,Z 579.319,A -85,B 0,C 180,E1 -1616.569,E2 -1616.569} C_VEL
LIN {X 0,Y 587.132,Z 581.196,A -85,B 0,C 180,E1 -1617.256,E2 -1617.256} C_VEL
LIN {X 0,Y 587.139,Z 582.628,A -85,B 0,C 180,E1 -1617.942,E2 -1617.942} C_VEL
LIN {X 0,Y 587.14,Z 584.254,A -85,B 0,C 180,E1 -1619.314,E2 -1619.314} C_VEL
LIN {X 0,Y 587.137,Z 584.496,A -85,B 0,C 180,E1 -1620,E2 -1620} C_VEL
LIN {X 0,Y 587.14,Z 584.315,A -85,B 0,C 180,E1 -1620.686,E2 -1620.686} C_VEL
LIN {X 0,Y 587.138,Z 582.774,A -85,B 0,C 180,E1 -1622.058,E2 -1622.058} C_VEL
LIN {X 0,Y 587.133,Z 581.413,A -85,B 0,C 180,E1 -1622.744,E2 -1622.744} C_VEL
LIN {X 0,Y 587.213,Z 578.536,A -85,B 0,C 180,E1 -1623.774,E2 -1623.774} C_VEL
LIN {X 0,Y 587.147,Z 574.636,A -85,B 0,C 180,E1 -1624.806,E2 -1624.806} C_VEL
LIN {X 0,Y 587.229,Z 569.604,A -85,B 0,C 180,E1 -1625.839,E2 -1625.839} C_VEL
LIN {X 0,Y 587.231,Z 563.283,A -85,B 0,C 180,E1 -1626.874,E2 -1626.874} C_VEL
LIN {X 0,Y 587.288,Z 555.364,A -85,B 0,C 180,E1 -1627.91,E2 -1627.91} C_VEL
LIN {X 0,Y 587.343,Z 545.517,A -85,B 0,C 180,E1 -1628.949,E2 -1628.949} C_VEL
LIN {X 0,Y 587.411,Z 535.195,A -85,B 0,C 180,E1 -1629.817,E2 -1629.817} C_VEL
LIN {X 0,Y 587.505,Z 523.567,A -85,B 0,C 180,E1 -1630.598,E2 -1630.598} C_VEL
LIN {X 0,Y 587.584,Z 512.701,A -85,B 0,C 180,E1 -1631.175,E2 -1631.175} C_VEL
LIN {X 0,Y 587.623,Z 499.946,A -85,B 0,C 180,E1 -1631.69,E2 -1631.69} C_VEL
LIN {X 0,Y 587.698,Z 486.986,A -85,B 0,C 180,E1 -1632.058,E2 -1632.058} C_VEL
LIN {X 0,Y 587.43,Z 480.901,A -85,B 0,C 180,E1 -1632.187,E2 -1632.187} C_VEL
LIN {X 0,Y 587.16,Z 479.214,A -85,B 0,C 180,E1 -1632.223,E2 -1632.223} C_VEL
LIN {X 0,Y 587.175,Z 476.924,A -85,B 0,C 180,E1 -1633.16,E2 -1633.16} C_VEL
LIN {X 0,Y 586.493,Z 475.606,A -85,B 0,C 180,E1 -1633.718,E2 -1633.718} C_VEL
LIN {X 0,Y 583.612,Z 473.582,A -85,B 0,C 180,E1 -1634.625,E2 -1634.625} C_VEL
LIN {X 0,Y 581.2,Z 471.982,A -85,B 0,C 180,E1 -1635.356,E2 -1635.356} C_VEL
LIN {X 0,Y 580.187,Z 470.706,A -85,B 0,C 180,E1 -1635.919,E2 -1635.919} C_VEL
LIN {X 0,Y 580.117,Z 470.259,A -85,B 0,C 180,E1 -1636.109,E2 -1636.109} C_VEL
LIN {X 0,Y 580.185,Z 463.223,A -85,B 0,C 180,E1 -1639.091,E2 -1639.091} C_VEL
LIN {X 0,Y 580.187,Z 456.355,A -85,B 0,C 180,E1 -1642.056,E2 -1642.056} C_VEL
LIN {X 0,Y 580.186,Z 449.486,A -85,B 0,C 180,E1 -1645.085,E2 -1645.085} C_VEL
LIN {X 0,Y 580.226,Z 443.435,A -85,B 0,C 180,E1 -1647.844,E2 -1647.844} C_VEL
LIN {X 0,Y 580.287,Z 437.485,A -85,B 0,C 180,E1 -1650.576,E2 -1650.576} C_VEL
LIN {X 0,Y 580.332,Z 431.661,A -85,B 0,C 180,E1 -1653.32,E2 -1653.32} C_VEL
LIN {X 0,Y 580.315,Z 426.827,A -85,B 0,C 180,E1 -1655.704,E2 -1655.704} C_VEL
LIN {X 0,Y 580.29,Z 426.829,A -85,B 0,C 180,E1 -1658.146,E2 -1658.146} C_VEL
LIN {X 0,Y 580.303,Z 426.828,A -85,B 0,C 180,E1 -1660.843,E2 -1660.843} C_VEL
LIN {X 0,Y 580.294,Z 426.829,A -85,B 0,C 180,E1 -1663.657,E2 -1663.657} C_VEL
LIN {X 0,Y 580.28,Z 426.83,A -85,B 0,C 180,E1 -1666.609,E2 -1666.609} C_VEL
LIN {X 0,Y 580.302,Z 426.828,A -85,B 0,C 180,E1 -1669.156,E2 -1669.156} C_VEL
LIN {X 0,Y 580.32,Z 426.891,A -85,B 0,C 180,E1 -1672.054,E2 -1672.054} C_VEL
LIN {X 0,Y 580.37,Z 433.212,A -85,B 0,C 180,E1 -1674.227,E2 -1674.227} C_VEL
LIN {X 0,Y 580.352,Z 441.145,A -85,B 0,C 180,E1 -1676.978,E2 -1676.978} C_VEL
LIN {X 0,Y 580.366,Z 449.366,A -85,B 0,C 180,E1 -1679.831,E2 -1679.831} C_VEL
LIN {X 0,Y 580.365,Z 455.934,A -85,B 0,C 180,E1 -1682.129,E2 -1682.129} C_VEL
LIN {X 0,Y 580.323,Z 463.635,A -85,B 0,C 180,E1 -1684.92,E2 -1684.92} C_VEL
LIN {X 0,Y 580.268,Z 471.116,A -85,B 0,C 180,E1 -1687.572,E2 -1687.572} C_VEL
LIN {X 0,Y 580.238,Z 479.667,A -85,B 0,C 180,E1 -1690.543,E2 -1690.543} C_VEL
LIN {X 0,Y 580.161,Z 488.271,A -85,B 0,C 180,E1 -1693.478,E2 -1693.478} C_VEL
LIN {X 0,Y 580.166,Z 493.309,A -85,B 0,C 180,E1 -1695.138,E2 -1695.138} C_VEL
LIN {X 0,Y 581.141,Z 498.381,A -85,B 0,C 180,E1 -1695.242,E2 -1695.242} C_VEL
LIN {X 0,Y 581.061,Z 512.684,A -85,B 0,C 180,E1 -1695.55,E2 -1695.55} C_VEL
LIN {X 0,Y 580.913,Z 526.523,A -85,B 0,C 180,E1 -1695.997,E2 -1695.997} C_VEL
LIN {X 0,Y 580.835,Z 538.917,A -85,B 0,C 180,E1 -1696.53,E2 -1696.53} C_VEL
LIN {X 0,Y 580.694,Z 550.46,A -85,B 0,C 180,E1 -1697.15,E2 -1697.15} C_VEL
LIN {X 0,Y 580.591,Z 562.552,A -85,B 0,C 180,E1 -1697.947,E2 -1697.947} C_VEL
LIN {X 0,Y 580.447,Z 573.488,A -85,B 0,C 180,E1 -1698.829,E2 -1698.829} C_VEL
LIN {X 0,Y 580.381,Z 582.635,A -85,B 0,C 180,E1 -1699.71,E2 -1699.71} C_VEL
LIN {X 0,Y 580.296,Z 591.825,A -85,B 0,C 180,E1 -1700.765,E2 -1700.765} C_VEL
LIN {X 0,Y 580.194,Z 599.495,A -85,B 0,C 180,E1 -1701.816,E2 -1701.816} C_VEL
LIN {X 0,Y 580.143,Z 606.824,A -85,B 0,C 180,E1 -1703.041,E2 -1703.041} C_VEL
LIN {X 0,Y 580.128,Z 613.378,A -85,B 0,C 180,E1 -1704.438,E2 -1704.438} C_VEL
LIN {X 0,Y 580.105,Z 617.222,A -85,B 0,C 180,E1 -1705.483,E2 -1705.483} C_VEL
LIN {X 0,Y 580.108,Z 620.205,A -85,B 0,C 180,E1 -1706.526,E2 -1706.526} C_VEL
LIN {X 0,Y 580.039,Z 622.912,A -85,B 0,C 180,E1 -1707.916,E2 -1707.916} C_VEL
LIN {X 0,Y 580.036,Z 624.295,A -85,B 0,C 180,E1 -1709.305,E2 -1709.305} C_VEL
LIN {X 0,Y 580.037,Z 624.354,A -85,B 0,C 180,E1 -1710.693,E2 -1710.693} C_VEL
LIN {X 0,Y 580.038,Z 623.052,A -85,B 0,C 180,E1 -1712.082,E2 -1712.082} C_VEL
LIN {X 0,Y 580.108,Z 620.429,A -85,B 0,C 180,E1 -1713.472,E2 -1713.472} C_VEL
LIN {X 0,Y 580.046,Z 616.372,A -85,B 0,C 180,E1 -1714.864,E2 -1714.864} C_VEL
LIN {X 0,Y 580.137,Z 612.33,A -85,B 0,C 180,E1 -1715.909,E2 -1715.909} C_VEL
LIN {X 0,Y 580.141,Z 607.3,A -85,B 0,C 180,E1 -1716.957,E2 -1716.957} C_VEL
LIN {X 0,Y 580.192,Z 600.102,A -85,B 0,C 180,E1 -1718.182,E2 -1718.182} C_VEL
LIN {X 0,Y 580.284,Z 592.55,A -85,B 0,C 180,E1 -1719.233,E2 -1719.233} C_VEL
LIN {X 0,Y 580.346,Z 583.482,A -85,B 0,C 180,E1 -1720.289,E2 -1720.289} C_VEL
LIN {X 0,Y 580.492,Z 572.55,A -85,B 0,C 180,E1 -1721.345,E2 -1721.345} C_VEL
LIN {X 0,Y 580.582,Z 561.329,A -85,B 0,C 180,E1 -1722.229,E2 -1722.229} C_VEL
LIN {X 0,Y 580.697,Z 549,A -85,B 0,C 180,E1 -1723.026,E2 -1723.026} C_VEL
LIN {X 0,Y 580.855,Z 537.159,A -85,B 0,C 180,E1 -1723.646,E2 -1723.646} C_VEL
LIN {X 0,Y 580.956,Z 522.578,A -85,B 0,C 180,E1 -1724.235,E2 -1724.235} C_VEL
LIN {X 0,Y 581.081,Z 508.762,A -85,B 0,C 180,E1 -1724.636,E2 -1724.636} C_VEL
LIN {X 0,Y 580.92,Z 497.143,A -85,B 0,C 180,E1 -1724.874,E2 -1724.874} C_VEL
LIN {X 0,Y 580.158,Z 493.167,A -85,B 0,C 180,E1 -1724.961,E2 -1724.961} C_VEL
LIN {X 0,Y 580.197,Z 484.211,A -85,B 0,C 180,E1 -1727.991,E2 -1727.991} C_VEL
LIN {X 0,Y 580.236,Z 476.725,A -85,B 0,C 180,E1 -1730.563,E2 -1730.563} C_VEL
LIN {X 0,Y 580.298,Z 468.169,A -85,B 0,C 180,E1 -1733.556,E2 -1733.556} C_VEL
LIN {X 0,Y 580.363,Z 459.613,A -85,B 0,C 180,E1 -1736.618,E2 -1736.618} C_VEL
LIN {X 0,Y 580.419,Z 452.092,A -85,B 0,C 180,E1 -1739.33,E2 -1739.33} C_VEL
LIN {X 0,Y 580.331,Z 443.798,A -85,B 0,C 180,E1 -1742.197,E2 -1742.197} C_VEL
LIN {X 0,Y 580.384,Z 436.618,A -85,B 0,C 180,E1 -1744.688,E2 -1744.688} C_VEL
LIN {X 0,Y 580.399,Z 427.976,A -85,B 0,C 180,E1 -1747.666,E2 -1747.666} C_VEL
LIN {X 0,Y 580.34,Z 426.821,A -85,B 0,C 180,E1 -1748.141,E2 -1748.141} C_VEL
LIN {X 0,Y 580.296,Z 426.83,A -85,B 0,C 180,E1 -1750.842,E2 -1750.842} C_VEL
LIN {X 0,Y 580.282,Z 426.825,A -85,B 0,C 180,E1 -1753.656,E2 -1753.656} C_VEL
LIN {X 0,Y 580.286,Z 426.826,A -85,B 0,C 180,E1 -1756.607,E2 -1756.607} C_VEL
LIN {X 0,Y 580.295,Z 426.825,A -85,B 0,C 180,E1 -1759.156,E2 -1759.156} C_VEL
LIN {X 0,Y 580.284,Z 426.825,A -85,B 0,C 180,E1 -1761.926,E2 -1761.926} C_VEL
LIN {X 0,Y 580.298,Z 426.826,A -85,B 0,C 180,E1 -1764.456,E2 -1764.456} C_VEL
LIN {X 0,Y 580.286,Z 426.826,A -85,B 0,C 180,E1 -1766.975,E2 -1766.975} C_VEL
LIN {X 0,Y 580.302,Z 426.822,A -85,B 0,C 180,E1 -1769.425,E2 -1769.425} C_VEL
LIN {X 0,Y 580.311,Z 426.822,A -85,B 0,C 180,E1 -1772.136,E2 -1772.136} C_VEL
LIN {X 0,Y 580.3,Z 426.826,A -85,B 0,C 180,E1 -1774.92,E2 -1774.92} C_VEL
LIN {X 0,Y 580.321,Z 426.822,A -85,B 0,C 180,E1 -1777.199,E2 -1777.199} C_VEL
LIN {X 0,Y 580.3,Z 426.826,A -85,B 0,C 180,E1 -1780.177,E2 -1780.177} C_VEL
LIN {X 0,Y 580.32,Z 426.82,A -85,B 0,C 180,E1 -1783.103,E2 -1783.103} C_VEL
LIN {X 0,Y 580.317,Z 426.822,A -85,B 0,C 180,E1 -1785.983,E2 -1785.983} C_VEL
LIN {X 0,Y 580.321,Z 426.823,A -85,B 0,C 180,E1 -1788.827,E2 -1788.827} C_VEL
LIN {X 0,Y 580.328,Z 426.818,A -85,B 0,C 180,E1 -1791.644,E2 -1791.644} C_VEL
LIN {X 0,Y 580.328,Z 426.823,A -85,B 0,C 180,E1 -1794.44,E2 -1794.44} C_VEL
LIN {X 0,Y 580.339,Z 426.819,A -85,B 0,C 180,E1 -1797.223,E2 -1797.223} C_VEL
LIN {X 0,Y 580.342,Z 426.818,A -85,B 0,C 180,E1 -1800,E2 -1800} C_VEL
LIN {X 0,Y 580.341,Z 426.822,A -85,B 0,C 180,E1 -1802.776,E2 -1802.776} C_VEL
LIN {X 0,Y 580.32,Z 426.819,A -85,B 0,C 180,E1 -1805.56,E2 -1805.56} C_VEL
LIN {X 0,Y 580.329,Z 426.822,A -85,B 0,C 180,E1 -1808.356,E2 -1808.356} C_VEL
LIN {X 0,Y 580.322,Z 426.819,A -85,B 0,C 180,E1 -1811.208,E2 -1811.208} C_VEL
LIN {X 0,Y 580.305,Z 426.822,A -85,B 0,C 180,E1 -1814.339,E2 -1814.339} C_VEL
LIN {X 0,Y 580.306,Z 426.824,A -85,B 0,C 180,E1 -1816.916,E2 -1816.916} C_VEL
LIN {X 0,Y 580.301,Z 426.824,A -85,B 0,C 180,E1 -1819.822,E2 -1819.822} C_VEL
LIN {X 0,Y 580.271,Z 426.832,A -85,B 0,C 180,E1 -1822.053,E2 -1822.053} C_VEL
LIN {X 0,Y 580.299,Z 426.825,A -85,B 0,C 180,E1 -1825.08,E2 -1825.08} C_VEL
LIN {X 0,Y 580.311,Z 426.821,A -85,B 0,C 180,E1 -1827.864,E2 -1827.864} C_VEL
LIN {X 0,Y 580.292,Z 426.83,A -85,B 0,C 180,E1 -1830.698,E2 -1830.698} C_VEL
LIN {X 0,Y 580.299,Z 426.822,A -85,B 0,C 180,E1 -1833.318,E2 -1833.318} C_VEL
LIN {X 0,Y 580.319,Z 426.827,A -85,B 0,C 180,E1 -1835.768,E2 -1835.768} C_VEL
LIN {X 0,Y 580.282,Z 426.825,A -85,B 0,C 180,E1 -1838.147,E2 -1838.147} C_VEL
LIN {X 0,Y 580.314,Z 426.826,A -85,B 0,C 180,E1 -1840.842,E2 -1840.842} C_VEL
LIN {X 0,Y 580.284,Z 426.824,A -85,B 0,C 180,E1 -1843.657,E2 -1843.657} C_VEL
LIN {X 0,Y 580.271,Z 426.828,A -85,B 0,C 180,E1 -1846.61,E2 -1846.61} C_VEL
LIN {X 0,Y 580.3,Z 426.824,A -85,B 0,C 180,E1 -1849.158,E2 -1849.158} C_VEL
LIN {X 0,Y 580.286,Z 426.826,A -85,B 0,C 180,E1 -1851.928,E2 -1851.928} C_VEL
LIN {X 0,Y 580.305,Z 426.825,A -85,B 0,C 180,E1 -1854.458,E2 -1854.458} C_VEL
LIN {X 0,Y 580.332,Z 426.938,A -85,B 0,C 180,E1 -1856.906,E2 -1856.906} C_VEL
LIN {X 0,Y 580.867,Z 430.389,A -85,B 0,C 180,E1 -1857.881,E2 -1857.881} C_VEL
LIN {X 0,Y 580.734,Z 440.946,A -85,B 0,C 180,E1 -1860.615,E2 -1860.615} C_VEL
LIN {X 0,Y 580.642,Z 452.012,A -85,B 0,C 180,E1 -1863.396,E2 -1863.396} C_VEL
LIN {X 0,Y 580.497,Z 462.94,A -85,B 0,C 180,E1 -1866.074,E2 -1866.074} C_VEL
LIN {X 0,Y 580.419,Z 474.304,A -85,B 0,C 180,E1 -1868.805,E2 -1868.805} C_VEL
LIN {X 0,Y 580.357,Z 487.917,A -85,B 0,C 180,E1 -1872.014,E2 -1872.014} C_VEL
LIN {X 0,Y 580.255,Z 501.089,A -85,B 0,C 180,E1 -1875.064,E2 -1875.064} C_VEL
LIN {X 0,Y 581.107,Z 505.695,A -85,B 0,C 180,E1 -1875.154,E2 -1875.154} C_VEL
LIN {X 0,Y 581.06,Z 520.095,A -85,B 0,C 180,E1 -1875.44,E2 -1875.44} C_VEL
LIN {X 0,Y 580.972,Z 534.658,A -85,B 0,C 180,E1 -1875.883,E2 -1875.883} C_VEL
LIN {X 0,Y 580.863,Z 548.117,A -85,B 0,C 180,E1 -1876.443,E2 -1876.443} C_VEL
LIN {X 0,Y 580.692,Z 561.276,A -85,B 0,C 180,E1 -1877.152,E2 -1877.152} C_VEL
LIN {X 0,Y 580.589,Z 573.159,A -85,B 0,C 180,E1 -1877.948,E2 -1877.948} C_VEL
LIN {X 0,Y 580.44,Z 584.003,A -85,B 0,C 180,E1 -1878.831,E2 -1878.831} C_VEL
LIN {X 0,Y 580.324,Z 594.716,A -85,B 0,C 180,E1 -1879.887,E2 -1879.887} C_VEL
LIN {X 0,Y 580.264,Z 603.567,A -85,B 0,C 180,E1 -1880.942,E2 -1880.942} C_VEL
LIN {X 0,Y 580.197,Z 612.044,A -85,B 0,C 180,E1 -1882.169,E2 -1882.169} C_VEL
LIN {X 0,Y 580.122,Z 618.994,A -85,B 0,C 180,E1 -1883.416,E2 -1883.416} C_VEL
LIN {X 0,Y 580.128,Z 623.572,A -85,B 0,C 180,E1 -1884.439,E2 -1884.439} C_VEL
LIN {X 0,Y 580.102,Z 628.445,A -85,B 0,C 180,E1 -1885.832,E2 -1885.832} C_VEL
LIN {X 0,Y 580.041,Z 631.833,A -85,B 0,C 180,E1 -1887.223,E2 -1887.223} C_VEL
LIN {X 0,Y 580.041,Z 633.833,A -85,B 0,C 180,E1 -1888.612,E2 -1888.612} C_VEL
LIN {X 0,Y 580.036,Z 634.5,A -85,B 0,C 180,E1 -1890.001,E2 -1890.001} C_VEL
LIN {X 0,Y 580.041,Z 633.831,A -85,B 0,C 180,E1 -1891.389,E2 -1891.389} C_VEL
LIN {X 0,Y 580.041,Z 631.831,A -85,B 0,C 180,E1 -1892.779,E2 -1892.779} C_VEL
LIN {X 0,Y 580.102,Z 628.441,A -85,B 0,C 180,E1 -1894.169,E2 -1894.169} C_VEL
LIN {X 0,Y 580.128,Z 623.564,A -85,B 0,C 180,E1 -1895.562,E2 -1895.562} C_VEL
LIN {X 0,Y 580.142,Z 617.048,A -85,B 0,C 180,E1 -1896.959,E2 -1896.959} C_VEL
LIN {X 0,Y 580.192,Z 609.794,A -85,B 0,C 180,E1 -1898.184,E2 -1898.184} C_VEL
LIN {X 0,Y 580.284,Z 600.816,A -85,B 0,C 180,E1 -1899.411,E2 -1899.411} C_VEL
LIN {X 0,Y 580.356,Z 591.383,A -85,B 0,C 180,E1 -1900.466,E2 -1900.466} C_VEL
LIN {X 0,Y 580.477,Z 581.308,A -85,B 0,C 180,E1 -1901.405,E2 -1901.405} C_VEL
LIN {X 0,Y 580.593,Z 569.419,A -85,B 0,C 180,E1 -1902.319,E2 -1902.319} C_VEL
LIN {X 0,Y 580.726,Z 556.634,A -85,B 0,C 180,E1 -1903.116,E2 -1903.116} C_VEL
LIN {X 0,Y 580.866,Z 544.142,A -85,B 0,C 180,E1 -1903.737,E2 -1903.737} C_VEL
LIN {X 0,Y 581.015,Z 531.165,A -85,B 0,C 180,E1 -1904.237,E2 -1904.237} C_VEL
LIN {X 0,Y 581.085,Z 517.146,A -85,B 0,C 180,E1 -1904.632,E2 -1904.632} C_VEL
LIN {X 0,Y 581.049,Z 505.492,A -85,B 0,C 180,E1 -1904.851,E2 -1904.851} C_VEL
LIN {X 0,Y 580.256,Z 500.983,A -85,B 0,C 180,E1 -1904.96,E2 -1904.96} C_VEL
LIN {X 0,Y 580.358,Z 487.909,A -85,B 0,C 180,E1 -1907.988,E2 -1907.988} C_VEL
LIN {X 0,Y 580.425,Z 474.296,A -85,B 0,C 180,E1 -1911.197,E2 -1911.197} C_VEL
LIN {X 0,Y 580.5,Z 462.932,A -85,B 0,C 180,E1 -1913.928,E2 -1913.928} C_VEL
LIN {X 0,Y 580.647,Z 452.004,A -85,B 0,C 180,E1 -1916.606,E2 -1916.606} C_VEL
LIN {X 0,Y 580.756,Z 440.989,A -85,B 0,C 180,E1 -1919.389,E2 -1919.389} C_VEL
LIN {X 0,Y 580.966,Z 430.639,A -85,B 0,C 180,E1 -1922.16,E2 -1922.16} C_VEL
LIN {X 0,Y 580.292,Z 426.831,A -85,B 0,C 180,E1 -1923.362,E2 -1923.362} C_VEL
LIN {X 0,Y 580.269,Z 426.832,A -85,B 0,C 180,E1 -1925.759,E2 -1925.759} C_VEL
LIN {X 0,Y 580.293,Z 426.826,A -85,B 0,C 180,E1 -1928.147,E2 -1928.147} C_VEL
LIN {X 0,Y 580.302,Z 426.826,A -85,B 0,C 180,E1 -1930.844,E2 -1930.844} C_VEL
LIN {X 0,Y 580.277,Z 426.83,A -85,B 0,C 180,E1 -1933.659,E2 -1933.659} C_VEL
LIN {X 0,Y 580.29,Z 426.829,A -85,B 0,C 180,E1 -1936.609,E2 -1936.609} C_VEL
LIN {X 0,Y 580.302,Z 426.829,A -85,B 0,C 180,E1 -1939.157,E2 -1939.157} C_VEL
LIN {X 0,Y 580.293,Z 426.829,A -85,B 0,C 180,E1 -1941.927,E2 -1941.927} C_VEL
LIN {X 0,Y 580.343,Z 426.959,A -85,B 0,C 180,E1 -1944.672,E2 -1944.672} C_VEL
LIN {X 0,Y 580.306,Z 431.972,A -85,B 0,C 180,E1 -1946.976,E2 -1946.976} C_VEL
LIN {X 0,Y 580.288,Z 437.321,A -85,B 0,C 180,E1 -1949.425,E2 -1949.425} C_VEL
LIN {X 0,Y 580.278,Z 443.299,A -85,B 0,C 180,E1 -1952.146,E2 -1952.146} C_VEL
LIN {X 0,Y 580.193,Z 449.285,A -85,B 0,C 180,E1 -1954.915,E2 -1954.915} C_VEL
LIN {X 0,Y 580.187,Z 456.149,A -85,B 0,C 180,E1 -1957.944,E2 -1957.944} C_VEL
LIN {X 0,Y 580.184,Z 463.013,A -85,B 0,C 180,E1 -1960.91,E2 -1960.91} C_VEL
LIN {X 0,Y 580.122,Z 469.878,A -85,B 0,C 180,E1 -1963.821,E2 -1963.821} C_VEL
LIN {X 0,Y 580.135,Z 475.027,A -85,B 0,C 180,E1 -1965.978,E2 -1965.978} C_VEL
LIN {X 0,Y 580.079,Z 479.21,A -85,B 0,C 180,E1 -1967.715,E2 -1967.715} C_VEL
LIN {X 0,Y 580.78,Z 484.975,A -85,B 0,C 180,E1 -1967.841,E2 -1967.841} C_VEL
LIN {X 0,Y 580.697,Z 497.354,A -85,B 0,C 180,E1 -1968.171,E2 -1968.171} C_VEL
LIN {X 0,Y 580.579,Z 510.379,A -85,B 0,C 180,E1 -1968.673,E2 -1968.673} C_VEL
LIN {X 0,Y 580.537,Z 522.048,A -85,B 0,C 180,E1 -1969.273,E2 -1969.273} C_VEL
LIN {X 0,Y 580.438,Z 532.829,A -85,B 0,C 180,E1 -1969.976,E2 -1969.976} C_VEL
LIN {X 0,Y 580.333,Z 542.604,A -85,B 0,C 180,E1 -1970.766,E2 -1970.766} C_VEL
LIN {X 0,Y 580.264,Z 551.496,A -85,B 0,C 180,E1 -1971.643,E2 -1971.643} C_VEL
LIN {X 0,Y 580.206,Z 560.18,A -85,B 0,C 180,E1 -1972.693,E2 -1972.693} C_VEL
LIN {X 0,Y 580.137,Z 567.107,A -85,B 0,C 180,E1 -1973.741,E2 -1973.741} C_VEL
LIN {X 0,Y 580.086,Z 572.657,A -85,B 0,C 180,E1 -1974.787,E2 -1974.787} C_VEL
LIN {X 0,Y 580.105,Z 577.018,A -85,B 0,C 180,E1 -1975.832,E2 -1975.832} C_VEL
LIN {X 0,Y 580.124,Z 579.321,A -85,B 0,C 180,E1 -1976.527,E2 -1976.527} C_VEL
LIN {X 0,Y 580.043,Z 581.198,A -85,B 0,C 180,E1 -1977.222,E2 -1977.222} C_VEL
LIN {X 0,Y 580.038,Z 582.628,A -85,B 0,C 180,E1 -1977.917,E2 -1977.917} C_VEL
LIN {X 0,Y 580.041,Z 584.254,A -85,B 0,C 180,E1 -1979.306,E2 -1979.306} C_VEL
LIN {X 0,Y 580.038,Z 584.496,A -85,B 0,C 180,E1 -1980,E2 -1980} C_VEL
LIN {X 0,Y 580.04,Z 584.315,A -85,B 0,C 180,E1 -1980.694,E2 -1980.694} C_VEL
LIN {X 0,Y 580.037,Z 582.772,A -85,B 0,C 180,E1 -1982.083,E2 -1982.083} C_VEL
LIN {X 0,Y 580.044,Z 581.411,A -85,B 0,C 180,E1 -1982.778,E2 -1982.778} C_VEL
LIN {X 0,Y 580.11,Z 578.534,A -85,B 0,C 180,E1 -1983.821,E2 -1983.821} C_VEL
LIN {X 0,Y 580.054,Z 574.633,A -85,B 0,C 180,E1 -1984.865,E2 -1984.865} C_VEL
LIN {X 0,Y 580.161,Z 569.601,A -85,B 0,C 180,E1 -1985.91,E2 -1985.91} C_VEL
LIN {X 0,Y 580.158,Z 563.279,A -85,B 0,C 180,E1 -1986.958,E2 -1986.958} C_VEL
LIN {X 0,Y 580.241,Z 555.359,A -85,B 0,C 180,E1 -1988.007,E2 -1988.007} C_VEL
LIN {X 0,Y 580.308,Z 545.511,A -85,B 0,C 180,E1 -1989.058,E2 -1989.058} C_VEL
LIN {X 0,Y 580.41,Z 535.188,A -85,B 0,C 180,E1 -1989.936,E2 -1989.936} C_VEL
LIN {X 0,Y 580.504,Z 523.556,A -85,B 0,C 180,E1 -1990.728,E2 -1990.728} C_VEL
LIN {X 0,Y 580.613,Z 512.004,A -85,B 0,C 180,E1 -1991.343,E2 -1991.343} C_VEL
LIN {X 0,Y 580.685,Z 500.121,A -85,B 0,C 180,E1 -1991.825,E2 -1991.825} C_VEL
LIN {X 0,Y 580.781,Z 486.962,A -85,B 0,C 180,E1 -1992.204,E2 -1992.204} C_VEL
LIN {X 0,Y 580.569,Z 482.327,A -85,B 0,C 180,E1 -1992.305,E2 -1992.305} C_VEL
LIN {X 0,Y 580.096,Z 479.213,A -85,B 0,C 180,E1 -1992.374,E2 -1992.374} C_VEL
LIN {X 0,Y 580.126,Z 473.525,A -85,B 0,C 180,E1 -1994.739,E2 -1994.739} C_VEL
LIN {X 0,Y 580.117,Z 470.259,A -85,B 0,C 180,E1 -1996.109,E2 -1996.109} C_VEL
LIN {X 0,Y 579.474,Z 468.962,A -85,B 0,C 180,E1 -1996.674,E2 -1996.674} C_VEL
LIN {X 0,Y 576.602,Z 467.001,A -85,B 0,C 180,E1 -1997.594,E2 -1997.594} C_VEL
LIN {X 0,Y 574.17,Z 465.455,A -85,B 0,C 180,E1 -1998.335,E2 -1998.335} C_VEL
LIN {X 0,Y 573.142,Z 464.211,A -85,B 0,C 180,E1 -1998.906,E2 -1998.906} C_VEL
LIN {X 0,Y 573.069,Z 463.772,A -85,B 0,C 180,E1 -1999.099,E2 -1999.099} C_VEL
LIN {X 0,Y 573.094,Z 458.071,A -85,B 0,C 180,E1 -2001.586,E2 -2001.586} C_VEL
LIN {X 0,Y 573.148,Z 451.202,A -85,B 0,C 180,E1 -2004.64,E2 -2004.64} C_VEL
LIN {X 0,Y 573.157,Z 446.134,A -85,B 0,C 180,E1 -2006.981,E2 -2006.981} C_VEL
LIN {X 0,Y 573.221,Z 440.702,A -85,B 0,C 180,E1 -2009.483,E2 -2009.483} C_VEL
LIN {X 0,Y 573.262,Z 434.898,A -85,B 0,C 180,E1 -2012.229,E2 -2012.229} C_VEL
LIN {X 0,Y 573.296,Z 429.59,A -85,B 0,C 180,E1 -2014.779,E2 -2014.779} C_VEL
LIN {X 0,Y 573.289,Z 427.702,A -85,B 0,C 180,E1 -2015.785,E2 -2015.785} C_VEL
LIN {X 0,Y 573.243,Z 427.707,A -85,B 0,C 180,E1 -2018.702,E2 -2018.702} C_VEL
LIN {X 0,Y 573.258,Z 427.706,A -85,B 0,C 180,E1 -2021.595,E2 -2021.595} C_VEL
LIN {X 0,Y 573.245,Z 427.706,A -85,B 0,C 180,E1 -2024.333,E2 -2024.333} C_VEL
LIN {X 0,Y 573.244,Z 427.708,A -85,B 0,C 180,E1 -2027.358,E2 -2027.358} C_VEL
LIN {X 0,Y 573.251,Z 427.708,A -85,B 0,C 180,E1 -2030.393,E2 -2030.393} C_VEL
LIN {X 0,Y 573.293,Z 427.832,A -85,B 0,C 180,E1 -2032.006,E2 -2032.006} C_VEL
LIN {X 0,Y 573.355,Z 433.633,A -85,B 0,C 180,E1 -2033.999,E2 -2033.999} C_VEL
LIN {X 0,Y 573.332,Z 441.984,A -85,B 0,C 180,E1 -2036.941,E2 -2036.941} C_VEL
LIN {X 0,Y 573.327,Z 450.215,A -85,B 0,C 180,E1 -2039.828,E2 -2039.828} C_VEL
LIN {X 0,Y 573.304,Z 458.264,A -85,B 0,C 180,E1 -2042.631,E2 -2042.631} C_VEL
LIN {X 0,Y 573.282,Z 465.774,A -85,B 0,C 180,E1 -2045.366,E2 -2045.366} C_VEL
LIN {X 0,Y 573.226,Z 474.324,A -85,B 0,C 180,E1 -2048.418,E2 -2048.418} C_VEL
LIN {X 0,Y 573.158,Z 482.875,A -85,B 0,C 180,E1 -2051.408,E2 -2051.408} C_VEL
LIN {X 0,Y 573.097,Z 491.426,A -85,B 0,C 180,E1 -2054.347,E2 -2054.347} C_VEL
LIN {X 0,Y 573.086,Z 493.348,A -85,B 0,C 180,E1 -2054.951,E2 -2054.951} C_VEL
LIN {X 0,Y 574.292,Z 499.749,A -85,B 0,C 180,E1 -2055.085,E2 -2055.085} C_VEL
LIN {X 0,Y 574.182,Z 514.473,A -85,B 0,C 180,E1 -2055.424,E2 -2055.424} C_VEL
LIN {X 0,Y 573.998,Z 528.77,A -85,B 0,C 180,E1 -2055.915,E2 -2055.915} C_VEL
LIN {X 0,Y 573.904,Z 540.721,A -85,B 0,C 180,E1 -2056.455,E2 -2056.455} C_VEL
LIN {X 0,Y 573.714,Z 553.397,A -85,B 0,C 180,E1 -2057.171,E2 -2057.171} C_VEL
LIN {X 0,Y 573.535,Z 566.05,A -85,B 0,C 180,E1 -2058.065,E2 -2058.065} C_VEL
LIN {X 0,Y 573.453,Z 576.302,A -85,B 0,C 180,E1 -2058.952,E2 -2058.952} C_VEL
LIN {X 0,Y 573.276,Z 585.883,A -85,B 0,C 180,E1 -2059.938,E2 -2059.938} C_VEL
LIN {X 0,Y 573.191,Z 594.563,A -85,B 0,C 180,E1 -2061.005,E2 -2061.005} C_VEL
LIN {X 0,Y 573.113,Z 602.828,A -85,B 0,C 180,E1 -2062.247,E2 -2062.247} C_VEL
LIN {X 0,Y 573.036,Z 609.199,A -85,B 0,C 180,E1 -2063.427,E2 -2063.427} C_VEL
LIN {X 0,Y 573,Z 614.766,A -85,B 0,C 180,E1 -2064.721,E2 -2064.721} C_VEL
LIN {X 0,Y 573.029,Z 618.292,A -85,B 0,C 180,E1 -2065.779,E2 -2065.779} C_VEL
LIN {X 0,Y 572.957,Z 621.745,A -85,B 0,C 180,E1 -2067.187,E2 -2067.187} C_VEL
LIN {X 0,Y 572.944,Z 623.789,A -85,B 0,C 180,E1 -2068.593,E2 -2068.593} C_VEL
LIN {X 0,Y 572.937,Z 624.468,A -85,B 0,C 180,E1 -2069.999,E2 -2069.999} C_VEL
LIN {X 0,Y 572.941,Z 623.862,A -85,B 0,C 180,E1 -2071.405,E2 -2071.405} C_VEL
LIN {X 0,Y 572.954,Z 621.932,A -85,B 0,C 180,E1 -2072.811,E2 -2072.811} C_VEL
LIN {X 0,Y 573.03,Z 618.568,A -85,B 0,C 180,E1 -2074.219,E2 -2074.219} C_VEL
LIN {X 0,Y 573.001,Z 615.123,A -85,B 0,C 180,E1 -2075.277,E2 -2075.277} C_VEL
LIN {X 0,Y 573.043,Z 609.599,A -85,B 0,C 180,E1 -2076.579,E2 -2076.579} C_VEL
LIN {X 0,Y 573.126,Z 602.334,A -85,B 0,C 180,E1 -2077.928,E2 -2077.928} C_VEL
LIN {X 0,Y 573.219,Z 593.905,A -85,B 0,C 180,E1 -2079.17,E2 -2079.17} C_VEL
LIN {X 0,Y 573.303,Z 585.096,A -85,B 0,C 180,E1 -2080.238,E2 -2080.238} C_VEL
LIN {X 0,Y 573.437,Z 575.88,A -85,B 0,C 180,E1 -2081.178,E2 -2081.178} C_VEL
LIN {X 0,Y 573.583,Z 564.924,A -85,B 0,C 180,E1 -2082.111,E2 -2082.111} C_VEL
LIN {X 0,Y 573.726,Z 551.996,A -85,B 0,C 180,E1 -2083.007,E2 -2083.007} C_VEL
LIN {X 0,Y 573.89,Z 540.753,A -85,B 0,C 180,E1 -2083.634,E2 -2083.634} C_VEL
LIN {X 0,Y 573.992,Z 528.804,A -85,B 0,C 180,E1 -2084.174,E2 -2084.174} C_VEL
